# B&R Automation Studio project PLC code - cp (part 18)

#### MachineCtrl_Slow.st - Calling program actions
```iecst
PROGRAM _INIT

	versionPLC;

	IF gPLC.iVersion0<>gPermanentVersion.iVersion0 OR gPLC.iVersion1<>gPermanentVersion.iVersion1 OR gPLC.iVersion2<>gPermanentVersion.iVersion2 THEN
		gMachine.AutoCmd.xCleanModbus := TRUE;
	END_IF

	PLC_Init(ADR(gPLC));

END_PROGRAM

PROGRAM _CYCLIC

	// ACTIONS
	InternalPLC;

	VarsVersion;

	// Manage resetting PLC
	resetPLC;

	//Setting Serial Name of the PLC
	setSerialNumber;

	GeneralMachineData;

	//Devices parameters assignation not required to be executed in fast cycle
	OrdersPrinterSlow;

	// It allows CleanBelt action integrated on BeltManager
	IF gMachine.Pt.Clean.xCleanBeltWater THEN
		CleanBeltWater; //NOZOMITWO-1912
	ELSIF NOT gMachine.Pt.Clean.xCleanBeltForUv THEN
		CleanBelt;
	ELSE
		IF gMachine.Pt.MachineModel<>Type_CUBE AND gMachine.Pt.MachineModel<>Type_CUBE_GULLIVER AND gMachine.Pt.MachineModel<>Type_CUBE_INSPECTION AND gMachine.Pt.MachineModel<>Type_CUBE_GULLIVER_INSPECTION  THEN
			CleanBeltUv;
		END_IF
	END_IF

	//
	CleanBeltTop;

	// It allows to have consent line in belt orders
	//[RGP] Execute "ConsentsLine" always. It was previously called if "gBelt.parameters.xExistConsentLine" was active and always was
	ConsentsLine;

	// TOJMH: Review loop
	CleanSystem;

	BeltShot;

	PowerCtrl;
	SuctionBlower;
	ResetRouterAndCB;

	AirCleaner;

	AlarmsSlow;

	IF gMachine.Pt.MachineLights = MACHINE_LIGHTS_RGB THEN
		RgbLigths;
	ELSE
		LightBeacon;
	END_IF

	//[RGP] Execution of this action not conditioned to "xControlledByLine" so line has not to manage buzzer conditions defined inside printer as referencing block, starting belt...
	SoundBeacon;
	Air;
	JamSensors;

	ProgramsManager;

	Remote;

	// Check coherency of values and log possible mismatches
	CheckValues;

	//  Hw activation. Always sending the information from Sw
	// now added a parameter indicating if it is dynamically allowed to enable the system or not
	gDing.Parameters.xEnable := gMachine.parSw.Hw.xInstallThicknessSensor;
	gPhotoCells.parameters.xEnable := gMachine.parSw.Hw.xInstallnSensor;

	Startup;

	gMachine.St.xStarted := TRUE;
	gMachine.St.exec.slow := gMachine.St.exec.slow +1;

	//Powermeter assignation
	gPowermeters[1].Inputs.Comms.ReceivedDataModPowerMeter := gReceivedDataModPowerMeter1;
	gPowermeters[2].Inputs.Comms.ReceivedDataModPowerMeter := gReceivedDataModPowerMeter2;

END_PROGRAM
```

#### VersionPLC.st
```iecst
ACTION versionPLC:

    // PLC Version
	gPLC.iVersion0 := 23;    // Major version
	gPLC.iVersion1 := 68;    // Refactoring
	gPLC.iVersion2 := 394;   // Updated ExtPack
	gPLC.iVersion3 := 563;   // Version

END_ACTION
```

#### VarsVersion.st
```iecst
// THIS CODE IS AUTOGENERATED. DO NOT MODIFY IT WITH AUTOMATION STUDIO
// Generation: 10/07/2024 16:17:34
// Program version: 2.1.4.0

ACTION VarsVersion:

	gPLC.iVarsVersion0 := 9;
	gPLC.iVarsVersion1 := 42;
	gPLC.iVarsVersion2 := 1;
	gPLC.iVarsVersion3 := 2;

END_ACTION
```

- InternalPLC.st (reference to Logical/Printer/MachineCtrl/MachineCtrl_Slow/InternalPLC.st)

#### GeneralMachineData.st - Constant values according machine model
```iecst
ACTION GeneralMachineData:

	//////////////////////////////////////////////////////////////////////////////////////////////////////////////////////
	// BELT PARAMS      BELT PARAMS      BELT PARAMS      BELT PARAMS      BELT PARAMS      BELT PARAMS      BELT PARAMS
	// BELT PARAMS      BELT PARAMS      BELT PARAMS      BELT PARAMS      BELT PARAMS      BELT PARAMS      BELT PARAMS
	//////////////////////////////////////////////////////////////////////////////////////////////////////////////////////

	// Cleaning Belt limits cannot be lower than 1
	// Cleaning Belt parameters. Clean Belt disabled/enabled after delay
	iSPTilesToCleanBelt		:= MAX (gMachine.parSw.CleanBelt.iSPTilesToCleanBelt, MIN_TILES_FOR_CLEANING_BELT);
	iSPTilesToCleanBeltTop	:= MAX (gMachine.parSw.CleanBeltTop.iSPTilesToCleanBelt, MIN_TILES_FOR_CLEANING_BELT_TOP);

	////////// Belt Limits //////////////////////////////////
	//[RGP] Sending speed setpoint to gBelt. Not assigned directly from SW so maybe in the future SpeedSetpoint need to be used outside BeltPackage/BeltManager.
	//As done in previous lines by limiting maximum belt speed. //Not been able to have a Zero value in the SetPointSpeed
	gMachine.parSw.Safety.rMaxBeltSpeedSetPoint := MAX(gMachine.parSw.Safety.rMaxBeltSpeedSetPoint, 20); //At least a minimum value of 20.0m/min as max value

	//Belt speed definition
	IF gLine.StatusSummary.xEmptyingBelts THEN
		gBelt.parameters.rSetPointSpeed := MIN(gMachine.Pt.rBeltSpeedWhileEmptyBelt, gMachine.parSw.rBeltSpeedSetPoint);

	ELSIF gMachine.St.CleaningBelt.xCleaningProcessOnGoing THEN
		gBelt.parameters.rSetPointSpeed := INT_TO_REAL(gMachine.parSw.CleanBelt.iBeltSpeed);

	ELSIF (gLine.Status <> LINE_CONTROLLED_STOP AND gLine.Status <> LINE_CLEANINGPH AND gLine.Status <> LINE_STARTING_CLEANINGPH) OR NOT gMachine.Pt.xControlledByLine THEN
		gBelt.parameters.rSetPointSpeed := gMachine.parSw.rBeltSpeedSetPoint;
	END_IF

	// It gets belt direction following if machine configuration is left or right
	gBelt.parameters.Direction:= NOT gMachine.parSw.xMachineDirection;

	//Appling physical limitations
	IF NOT gMachine.Pt.xControlledByLine THEN
		gBelt.parameters.rMaxSpeed := gBelt.states.Hw.rMaxSpeed;
		gMachine.St.xDoubleLineAllowed := gMachine.Pt.Hw.xDoubleLineAllowed AND NOT gEdgeHoldDown.status.xEnabled;

	ELSE
		gBelt.parameters.rMaxSpeed := MIN(gBelt.states.Hw.rMaxSpeed, gLine.Parameters.Hw.rMaxSpeed);
		gMachine.St.xDoubleLineAllowed := gMachine.Pt.Hw.xDoubleLineAllowed AND gLine.Parameters.Hw.xDoubleLineAllowed AND NOT gEdgeHoldDown.status.xEnabled;
	END_IF

	////////////////////////////////////////////////////////////////////////////////////////////////////////////
	// BLOCK
	////////////////////////////////////////////////////////////////////////////////////////////////////////////

	xAnyBlockToPrint:=FALSE;
	FOR iIndexBlock:=1 TO gMachine.Pt.CT.iNumBlocks DO
		// It is used by ModeActive	implemented on printer
		IF gBlock[iIndexBlock].parSw.xEnableToPrint THEN
			xAnyBlockToPrint:=TRUE;
		END_IF
	END_FOR
	gMachine.St.Blocks.xAnyBlockToPrint:=xAnyBlockToPrint;

	///////////
	//White
	///////////
	IF gMachine.St.White.xInstalled THEN
		//Defining white bar index depending on machine direction. White is always first mechanically installed print bar
		IF gMachine.parSw.xMachineDirection THEN
			iWhiteBarMechanicalPosition := gBlock[1].parameters.Inks.iMaxMachinePrintBars;
		ELSE
			iWhiteBarMechanicalPosition := 1;
		END_IF

		IF NOT gMachine.St.White.xDebugMode THEN
			gMachine.St.White.xEnableToPrint := gInks[iWhiteBarMapping].status.xColorLoadedInJob;
		END_IF
	ELSE
		gMachine.St.White.xEnableToPrint := FALSE;
	END_IF

	///////////
	//Clear
	///////////
	IF gMachine.St.Clear.xInstalled THEN
		//Defining Primer bar index depending on machine direction. Primer is always first mechanically installed print bar
		IF gMachine.parSw.xMachineDirection THEN
			iPrimerBarMechanicalPosition := 3;
		ELSE
			iPrimerBarMechanicalPosition := 8;
		END_IF

		IF NOT gMachine.St.Clear.xDebugMode THEN
			gMachine.St.Clear.xEnableToPrint := gInks[iPrimerBarMapping].status.xColorLoadedInJob;
		END_IF

	ELSE
		gMachine.St.Clear.xEnableToPrint := FALSE;
	END_IF

	///////////
	//Color
	///////////
	IF NOT gMachine.St.Color.xDebugMode THEN
		//DELOREAN-3427: In case no color bar is loaded in job, curing led bar type CURING_APP_COLOR wont be activated
		xColorBarEnabledToPrint:=FALSE;
		FOR iIndexInks:=1 TO MAX_LAST_INK DO
			IF iIndexInks<>iWhiteBarMapping AND iIndexInks<>iPrimerBarMapping THEN
				IF gInks[iIndexInks].status.xColorLoadedInJob THEN
					xColorBarEnabledToPrint:=TRUE;
					EXIT;
				END_IF
			END_IF
		END_FOR
		gMachine.St.Color.xEnableToPrint := xColorBarEnabledToPrint;
	END_IF

	//CUBE-1197: due to this issue, protecting curing process by enabling curingled bar in case there is only one curing led bar.
	IF gMachine.Pt.Hw.iMaxCuringLedBars=1 THEN
		gMachine.St.Color.xEnableToPrint:=iIndexColorCuringLedBar=1;
		gMachine.St.Clear.xEnableToPrint :=iIndexPrimerCuringLedBar=1; //Pending to change the name of "iIndexPrimerCuringLedBar" by "iIndexClearCuringLedBar"
		xWhiteBarEnabledToPrint:=iIndexWhiteCuringLedBar=1;
	END_IF

	////////////////////////////////////////////////////////////////////////////////////////////////////////////
	// INKS >>>>> SLOW FOR		SLOW FOR		SLOW FOR		SLOW FOR		SLOW FOR
	////////////////////////////////////////////////////////////////////////////////////////////////////////////

	// Reset the index if the index is not valid. Just for protection. Never should enter here
	IF iIndexInksSlow = 0 OR iIndexInksSlow > MAX_LAST_INK THEN
		StartValuesForInksSlowFor;
		iIndexInksSlow := 1;
	END_IF

	IF gInks[iIndexInksSlow].status.xInksRunning THEN
		xAnyInkBarStarted := TRUE;
		IF rMaxStartedTempSetPoint < gInks[iIndexInksSlow].parSw.Temp.rSetPointTemp THEN
			rMaxStartedTempSetPoint := gInks[iIndexInksSlow].parSw.Temp.rSetPointTemp;
		END_IF
		IF rMaxStartedInkTemp < gInks[iIndexInksSlow].status.Temp.rTemp THEN
			rMaxStartedInkTemp:= gInks[iIndexInksSlow].status.Temp.rTemp;
		END_IF
		IF rMinStartedTempSetPoint > gInks[iIndexInksSlow].parSw.Temp.rSetPointTemp THEN
			rMinStartedTempSetPoint := gInks[iIndexInksSlow].parSw.Temp.rSetPointTemp;
		END_IF
		IF rMinStartedInkTemp > gInks[iIndexInksSlow].status.Temp.rTemp THEN
			rMinStartedInkTemp:= gInks[iIndexInksSlow].status.Temp.rTemp;
		END_IF

		//Any Tank Enabled
		IF gInks[iIndexInksSlow].status.xInkAndPreheatingRunning THEN
			xAnyTankHeaterEnabled:= TRUE;
		END_IF

		//Any bar printhead enabled
		IF gInks[iIndexInksSlow].signals.out.xOutPowPrintHead THEN
			xAnyPrintheadsPowered:= TRUE;
		END_IF

		//Depending on white bar mechanical position and if its enabled to print by electronics, status variable is set.
		//Cannot assume that gInks[1] will be the white bar so there is a case were white is physically installed but not defined in printer UI (disabled), gInks[1] then would be the following print bar assembled
		IF gInks[iIndexInksSlow].parSw.Config.iMappingBar = iWhiteBarMechanicalPosition THEN
			iWhiteBarMapping := iIndexInksSlow;
		ELSIF gInks[iIndexInksSlow].parSw.Config.iMappingBar = iPrimerBarMechanicalPosition THEN
			iPrimerBarMapping := iIndexInksSlow;
		END_IF

		IF gInks[iIndexInksSlow].parameters.InksChiller.iIndex > 0 AND gInks[iIndexInksSlow].parameters.InksChiller.iIndex < MAX_LAST_CHILLER THEN // Adding safety in the assignation
			gInks[iIndexInksSlow].parameters.InksChiller.Status := gChiller[gInks[iIndexInksSlow].parameters.InksChiller.iIndex].St.Status;
		END_IF

	END_IF

	IF gInks[iIndexInksSlow].parameters.PrintheadsChiller.iIndex > 0 AND gInks[iIndexInksSlow].parameters.PrintheadsChiller.iIndex < MAX_LAST_CHILLER THEN //Adding safety in the assignation
		gInks[iIndexInksSlow].parameters.PrintheadsChiller.Status := gChiller[gInks[iIndexInksSlow].parameters.PrintheadsChiller.iIndex].St.Status;
	END_IF

	iIndexInksSlow := iIndexInksSlow + 1;

	//If there is no logical bar with the mapping of the physical position, reset the outputs
	IF iIndexInksSlow > MAX_LAST_INK THEN

		//Assign data calculated to Machine Data
		gMachine.St.Inks.xAnyStarted := xAnyInkBarStarted;
		gMachine.St.Inks.rMaxTempSetPoint := rMaxStartedTempSetPoint;
		gMachine.St.Inks.rMinTempSetPoint := rMinStartedTempSetPoint;
		gMachine.St.Inks.rMaxTemp := rMaxStartedInkTemp;
		gMachine.St.Inks.rMinTemp := rMinStartedInkTemp;

		gMachine.St.Blocks.xAnyTankHeaterEnabled:= xAnyTankHeaterEnabled;
		gMachine.St.Blocks.xAnyPrintheadPowered:= xAnyPrintheadsPowered;

		StartValuesForInksSlowFor;
		iIndexInksSlow := 1;
	END_IF

	// Jetting Gap limits
	gMachine.parSw.rMarginPrint:= LIMIT(gMachine.Pt.CT.rMinMarginPrinting,gMachine.parSw.rMarginPrint,gMachine.Pt.CT.rMaxMarginPrinting);

	// Piece Tickness
	gMachine.parSw.Media.rThickness:= LIMIT(gMachine.Pt.CT.rMinTicknessMedia,gMachine.parSw.Media.rThickness,gMachine.Pt.CT.rMaxTicknessMedia);

	// Mounted Tile
	gMachine.parSw.Safety.rMountedPieceOverthickness:= LIMIT(gMachine.Pt.CT.rMinMountedPieceOverThick,gMachine.parSw.Safety.rMountedPieceOverthickness,gMachine.Pt.CT.rMaxMountedPieceOverThick);

	// Cleaning by pieces
	gMachine.parSw.Clean.iPiecesNumberToCleanL1:= MAX (gMachine.parSw.Clean.iPiecesNumberToCleanL1, GC_MIN_PIECES_TO_CLEAN);
	gMachine.parSw.Clean.iPiecesNumberToCleanL2:= MAX (gMachine.parSw.Clean.iPiecesNumberToCleanL2, GC_MIN_PIECES_TO_CLEAN);

	// Counters of shots printed by PD or by simulation
	//Counting out of any FOR. Makes no sense
	IF EDGEPOS (gMachine.St.ProductDetect.xProductDetectL1) THEN
		gMachine.Lg.udiPiecesCounterL1:= gMachine.Lg.udiPiecesCounterL1 + 1;
	END_IF

	IF EDGEPOS (gMachine.St.ProductDetect.xProductDetectL2) THEN
		gMachine.Lg.udiPiecesCounterL2:= gMachine.Lg.udiPiecesCounterL2 + 1;
	END_IF

	gMachine.St.xWorkingAsPBF := gMachine.parSw.Electronics.xIsPBF;

	//When entering in Working as PBF, modify diPiecesCounterStrobe to keep the same quantity of differences
	IF EDGEPOS(gMachine.St.xWorkingAsPBF) THEN
		gMachine.Lg.diPiecesCounterStrobe := gMachine.Lg.udiPiecesCounterL1 - gMachine.Lg.iDiffPiecesStrobeProductDetect;
	END_IF

	//Count strobes when Bit8 (strobe) is actived
	IF EDGEPOS(gMachine.In.iRelieve1>=256) AND gMachine.St.xWorkingAsPBF THEN
		gMachine.Lg.diPiecesCounterStrobe:= gMachine.Lg.diPiecesCounterStrobe + 1;
		gMachine.Out.iRelief1 := gMachine.In.iRelieve1;
	END_IF

	//Remove Relief output after time enough for the kernel to read it
	tofKeepReliefSignal.IN := EDGEPOS(gMachine.In.iRelieve1>=256) AND gMachine.St.xWorkingAsPBF;
	tofKeepReliefSignal.PT := t#900ms;
	tofKeepReliefSignal();
	IF NOT tofKeepReliefSignal.Q THEN
		gMachine.Out.iRelief1 := 0;
	END_IF

	//If Reset the counter, assign the value of Strobes to the value of PD
	IF gMachine.commands.xResetStrobePdDiff THEN
		gMachine.Lg.diPiecesCounterStrobe := gMachine.Lg.udiPiecesCounterL1;
		gMachine.Lg.iDiffPiecesStrobeProductDetect := 0;
		gMachine.commands.xResetStrobePdDiff := FALSE;
	END_IF
	IF EDGEPOS(gMachine.Lg.udiPiecesCounterL1 = 0) THEN
		gMachine.Lg.diPiecesCounterStrobe := - gMachine.Lg.iDiffPiecesStrobeProductDetect;
	END_IF

	//Define the diff counter. Updated just when receive a media in Product detect
	IF gMachine.St.xWorkingAsPBF AND EDGEPOS (gMachine.St.ProductDetect.xProductDetectL1) THEN
		gMachine.Lg.iDiffPiecesStrobeProductDetect := DINT_TO_INT(gMachine.Lg.udiPiecesCounterL1 - gMachine.Lg.diPiecesCounterStrobe);
	END_IF

	// Machine conversions
	gMachine.Lg.udiDifCounters:=ABS(UDINT_TO_INT(gMachine.Lg.udiPiecesCounterL1-gDing.State.diLgLowPieceCounter));

	//Enable degasser
	gMachine.Out.xDegasser:= gMachine.parSw.xDegasser AND NOT gMachine.Al.Warning.xAlrDegasserPressure;

	//Safety
	gSafetyController.Parameters.xSimulationMode := gMachine.Pt.ConfigNameID = GC_CONFIG_SIMTEST_ID;

	//Define a transmision data to do the first calculations and be receptive to next calculations
	DriveUnit.TransmissionData.TransmissionType := TRANS_LINEAL_PERIMETER;
	DriveUnit.TransmissionData.LinealPerimeter.PulsesPerTurn := GC_UNITS_BY_REV_DRIVE;
	DriveUnit.TransmissionData.LinealPerimeter.GearBox := 10.0;
	DriveUnit.TransmissionData.LinealPerimeter.Perimeter := 500.0;

	IF gThicknessCtrl.status.Belt.rBeltPositionMmInit<>rBeltPositionMmInitCopy THEN
		//Logger
		//Calculation of position when mounted media alarm is raised
		DriveUnit.pulsesDevice := gThicknessCtrl.status.Belt.rBeltPositionMmInit;
		DriveUnit.Calculation := CALC_POS_MM;
		DriveUnit();
		rBeltPositionMmInit := DriveUnit.PositionDevice;

		//Calculation of position when mounted media alarm is raised
		DriveUnit.PulsesSpeedDevice := gThicknessCtrl.status.Belt.rBeltSpeed;
		DriveUnit.Calculation := CALC_SPEED_MMIN;
		DriveUnit();
		rBeltSpeedInit := ABS(DriveUnit.SpeedMminDevice);

		rBeltPositionMmInitCopy := gThicknessCtrl.status.Belt.rBeltPositionMmInit;
	END_IF

	IF gThicknessCtrl.status.Belt.rBeltPositionMmFinal<>rBeltPositionMmFinalCopy THEN
		//Calculation of position when belt stops
		DriveUnit.pulsesDevice := gThicknessCtrl.status.Belt.rBeltPositionMmFinal;
		DriveUnit.Calculation := CALC_POS_MM;
		DriveUnit();
		rBeltPositionMmFinal := DriveUnit.PositionDevice;

		rBeltPositionMmFinalCopy := gThicknessCtrl.status.Belt.rBeltPositionMmFinal;
	END_IF

	rBeltDistanceTravelledMm := rBeltPositionMmFinal - rBeltPositionMmInit;
	IF rBeltDistanceTravelledMm<>rBeltDistanceTravelledMmCopy THEN
		//Logging distance run by belt from mounted media event to be stopped
		LogBeltDistanceTravelledWhenMountedMedia;

		rBeltDistanceTravelledMmCopy := rBeltDistanceTravelledMm;
	END_IF

END_ACTION

ACTION StartValuesForInksSlowFor:
	xAnyInkBarStarted := FALSE;
	rMaxStartedTempSetPoint := 0.0; //To be sure to be decreased
	rMaxStartedInkTemp := 0.0; //To be sure to be decreased
	rMinStartedTempSetPoint := 100.0; //To be sure to be decreased
	rMinStartedInkTemp := 100.0; //To be sure to be decreased
	xAnyTankHeaterEnabled := FALSE;
	xAnyPrintheadsPowered := FALSE;
END_ACTION
```

#### CleanBelt.st - Clean belt order
```iecst
ACTION CleanBelt:

	///////////////////////////////////////////////////////////////////////////////////////////////////////////////////
	// General conditions to clean belt	when machine is in AUTOMATIC OR MANUAL MODES
	///////////////////////////////////////////////////////////////////////////////////////////////////////////////////

	//Cleaning Belt by time. When cleaning, the time is reseted
	tonCleaningByTime.IN:= gBelt.states.xRuningBelt AND gMachine.parSw.CleanBelt.xCleanBeltByTime AND NOT tonCleaningByTime.Q AND NOT xCleanBeltOrder AND gMachine.St.Mode.xAuto;
	tonCleaningByTime.PT := MAX(gMachine.parSw.CleanBelt.tiCleaningBeltByTime, MIN_TIME_FOR_CLEANING_BELT); // Time converted from minutes to miliseconds
	tonCleaningByTime();

	//Delay falling the tray to be sure no water is poured inside the machine
	tofCleaningTrayBelt.IN:=xCleanBeltOrder;
	tofCleaningTrayBelt.PT:=T#200MS;
	tofCleaningTrayBelt();

	//Delay pneumatic pump to avoid pouring water inside the machine
	tonCleanBelt.IN:= xCleanBeltOrder;
	tonCleanBelt.PT:=T#900ms;
	tonCleanBelt();

	//If the belt is not running, it is not possible to clean it
	IF NOT gBelt.states.xRuningBelt THEN
		gMachine.commands.CleanBelt := ResetCleanBeltCommands;
		xCleanBeltOrder := FALSE;
		RETURN;
	END_IF

	// Tiles counter
	IF gMachine.parSw.CleanBelt.xCleanBeltByTiles AND (EDGEPOS (gMachine.St.ProductDetect.xProductDetectL1) OR EDGEPOS(gMachine.St.ProductDetect.xProductDetectL2)) THEN
		gMachine.Lg.iTilesCounterToClean:= gMachine.Lg.iTilesCounterToClean+1;
	END_IF

	//Cleaning by tiles. When cleaning, number of tiles is reseted
	IF (gMachine.parSw.CleanBelt.xCleanBeltByTiles AND (gMachine.Lg.iTilesCounterToClean >= INT_TO_UINT(iSPTilesToCleanBelt)) AND gMachine.St.Mode.xAuto) THEN
		xCleaningBeltByTiles:= TRUE;
	END_IF

	// Force cleaning applying delay. Why clean continuous is same that condition than force clean?
	IF gMachine.parSw.CleanBelt.xCleanBeltForced THEN
		xCleanBeltForced:= TRUE;
		gMachine.parSw.CleanBelt.xCleanBeltForced := FALSE;
	END_IF

	IF tonCleaningByTime.Q THEN
		xCleaningBeltByTime:=TRUE;
	END_IF

	IF (gMachine.parSw.CleanBelt.xCleanBeltContinue AND gMachine.St.Mode.xAuto) THEN
		xCleanBeltContinue := TRUE;
	ELSE
		xCleanBeltContinue := FALSE;
	END_IF

	IF xCleaningBeltByTiles OR xCleaningBeltByTime OR xCleanBeltForced OR xCleanBeltContinue THEN
		xCleanBeltOrder:=TRUE;

		//Removed orders when cleaning
		xCleaningBeltByTiles:=FALSE;
		gMachine.Lg.iTilesCounterToClean:=0;
		xCleaningBeltByTime:=FALSE;
		xCleanBeltForced := FALSE;
	END_IF

	// Managing the duration of the belt cleaning
	tonCleaningBelt.IN:= xCleanBeltOrder;
	tonCleaningBelt.PT := MAX(gMachine.parSw.CleanBelt.tiCleaningBeltDuration, MIN_DURATION_CLEANING_BELT);
	tonCleaningBelt();

	IF (tonCleaningBelt.Q AND NOT(xCleanBeltContinue)) OR EDGENEG(xCleanBeltContinue) THEN
		xCleanBeltOrder:=FALSE;
	END_IF

	//////////////////////
	// OUTPUT management
	//////////////////////
	//Clean belt

	//Pneumatic
	gMachine.commands.CleanBelt.xPistonFlojet := tofCleaningTrayBelt.Q;
	gMachine.commands.CleanBelt.xCleanBeltPump := tonCleanBelt.Q;

END_ACTION

ACTION CleanBeltTop:

	IF NOT gMachine.Pt.Clean.xCleanBeltTopInstall OR NOT gBelt.states.xRuningBelt THEN
		xCleanBeltTopOrder						:= FALSE;
		RETURN;
	END_IF

	///////////////////////////////////////////////////////////////////////////////////////////////////////////////////
	// General conditions to clean belt	when machine is in AUTOMATIC OR MANUAL MODES
	///////////////////////////////////////////////////////////////////////////////////////////////////////////////////

	//Cleaning Belt by time. When cleaning, the time is reseted
	tonCleanBeltTopByTime.IN := gMachine.parSw.CleanBeltTop.xCleanBeltByTime AND NOT tonCleanBeltTopByTime.Q AND NOT xCleanBeltTopOrder AND gMachine.St.Mode.xAuto;
	tonCleanBeltTopByTime.PT := MAX(gMachine.parSw.CleanBeltTop.tiCleaningBeltByTime, MIN_TIME_FOR_CLEANING_TOP_BELT);
	tonCleanBeltTopByTime();

	// Tiles counter
	IF gMachine.parSw.CleanBeltTop.xCleanBeltByTiles AND (EDGEPOS (gMachine.St.ProductDetect.xProductDetectL1) OR EDGEPOS(gMachine.St.ProductDetect.xProductDetectL2)) THEN
		gMachine.Lg.iTilesCounterToCleanBeltTop:= gMachine.Lg.iTilesCounterToCleanBeltTop + 1;
	END_IF

	//Cleaning by tiles. When cleaning, number of tiles is reseted
	IF (gMachine.parSw.CleanBeltTop.xCleanBeltByTiles AND (gMachine.Lg.iTilesCounterToCleanBeltTop >= INT_TO_UINT(iSPTilesToCleanBeltTop)) AND gMachine.St.Mode.xAuto) THEN
		xCleaningBeltTopByTiles:= TRUE;
	END_IF

	// Force cleaning applying delay. Why clean continuous is same that condition than force clean?
	IF gMachine.parSw.CleanBeltTop.xCleanBeltForced THEN
		xCleanBeltTopForced:= TRUE;
		gMachine.parSw.CleanBeltTop.xCleanBeltForced := FALSE;
	END_IF

	IF tonCleanBeltTopByTime.Q THEN
		xCleaningBeltTopByTime:=TRUE;
	END_IF

	IF (gMachine.parSw.CleanBeltTop.xCleanBeltContinue AND gMachine.St.Mode.xAuto) THEN
		xCleanBeltTopContinue := TRUE;
	ELSE
		xCleanBeltTopContinue := FALSE;
	END_IF

	IF xCleaningBeltTopByTiles OR xCleaningBeltTopByTime OR xCleanBeltTopForced OR xCleanBeltTopContinue THEN
		xCleanBeltTopOrder:=TRUE;

		//Removed orders when cleaning
		xCleaningBeltTopByTiles:=FALSE;
		gMachine.Lg.iTilesCounterToCleanBeltTop:=0;
		xCleaningBeltTopByTime:=FALSE;
		xCleanBeltTopForced := FALSE;
	END_IF

	// Managing the duration of the belt cleaning
	tonCleaningBeltTop.IN:= xCleanBeltTopOrder;
	tonCleaningBeltTop.PT := MAX(gMachine.parSw.CleanBeltTop.tiCleaningBeltDuration, MIN_DURATION_CLEANING_BELT_TOP);
	tonCleaningBeltTop();

	IF (tonCleaningBeltTop.Q AND NOT(gMachine.parSw.CleanBeltTop.xCleanBeltContinue)) OR EDGENEG(gMachine.parSw.CleanBeltTop.xCleanBeltContinue) THEN
		xCleanBeltTopOrder:=FALSE;
	END_IF

	//////////////////////
	// OUTPUT management
	//////////////////////

	gMachine.commands.CleanBelt.xCleanBeltTopScraper:=xCleanBeltTopOrder AND NOT gMachine.Pt.Clean.xCleanBeltForUv;

END_ACTION
```

#### ConsentLine.st - Consent Line
```iecst
ACTION ConsentsLine:
		(*
		View OF the machine from the Operator side

		>>>>>> LeftHandMachine 					RightHandMachine <<<<<<<<
		(BK_A #1 >> BK_B #2)		LOGICAL			(BK_A #2 << BK_B #1)

			          ################-################
		L2	          ################-################     L2
		------        ################-################   -------
		L1	          ################-################     L1
			##########################-###########################
			##########################-###########################
			    ######################-#######################
			    ######################-#######################
			    ######################-#######################
			    ######################-#######################

			BLOCK A [1-physical]				BLOCK B [2-physical]

		*)

	///////////////////////////////////////////////////
	// Consents depending if double or simple line
	//////////////////////////////////////////////////
	xDoubleLineConsent:= 	( gMachine.parSw.Dtp.iModeLine1=GC_DTP_STOP OR gMachine.In.xConsentL1Ok ) AND
							( gMachine.parSw.Dtp.iModeLine2=GC_DTP_STOP OR gMachine.In.xConsentL2Ok ) AND
							( gMachine.parSw.Dtp.iModeLine1<>GC_DTP_STOP OR gMachine.parSw.Dtp.iModeLine2<>GC_DTP_STOP);

	tonDelayConsentInput.IN:= 	(NOT gMachine.parSw.Dtp.xDoubleLine AND gMachine.In.xConsentL1Ok ) OR
								(gMachine.parSw.Dtp.xDoubleLine AND xDoubleLineConsent );
	tonDelayConsentInput.PT:= T#500ms;
	tonDelayConsentInput();

	gMachine.St.Consent.xConsent:= tonDelayConsentInput.Q;

	//Raise Bars without consent
	xAvoidRaiseBarsNotConsent := gMachine.Al.Alarm.xAlarmNotInPrintPosition OR gMachine.Al.Warning.xNotLoadedImage;
	tonUpBarsNoConsent.IN :=	gMachine.St.AutoMode.xProduction AND NOT xAvoidRaiseBarsNotConsent AND NOT gMachine.St.Consent.xConsent;
	tonUpBarsNoConsent.PT:= T#5m;
	tonUpBarsNoConsent();
	gMachine.St.Consent.xUpWithNoConsentCountingTime := tonUpBarsNoConsent.IN;

	//Split the assignation to allow an external assignation from simulation to avoid waiting 5min
	IF EDGEPOS(tonUpBarsNoConsent.Q) THEN
		gMachine.St.Consent.xUpWithNoConsent := TRUE;
	END_IF
	IF NOT gMachine.St.AutoMode.xProduction OR EDGEPOS(gMachine.St.Position.xInPrint) THEN
		gMachine.St.Consent.xUpWithNoConsent := FALSE;
	END_IF

	IF gMachine.St.Consent.xUpWithNoConsent OR gMachine.St.xProtectBendedWithPause THEN
		gMachine.St.Consent.xOrderToEmpyBelt := TRUE;
	ELSIF NOT gThicknessCtrl.status.MediaPosition.xMediaInside THEN
		gMachine.St.Consent.xOrderToEmpyBelt := FALSE;
	END_IF

	///////////////////////////////////////////////////////////////////////////////////////
	///////////////////////////////////////////////////////////////////////////////////////
	///////////////////////////////////////////////////////////////////////////////////////

	// Pending to test
	//Consent Outputs for L1
	//Single line L1, When belt is runing is because we had consent
	xOutputConsentInSingleLineL1:=	NOT gMachine.parSw.Dtp.xDoubleLine AND
									gMachine.In.xConsentL1Ok AND
									gMachine.St.AutoMode.xProdORByPass AND
									NOT gThicknessCtrl.status.MediaPosition.xMountedMediaInside AND
									NOT gMachine.St.Blocks.xBlockAlarmToEmpyBelt AND
									NOT gMachine.St.Consent.xOrderToEmpyBelt;

	xOutputConsentInByPassL1 := gMachine.St.AutoMode.xBypass AND
								gMachine.In.xConsentL1Ok AND
								(NOT gMachine.parSw.Dtp.xDoubleLine OR (gMachine.parSw.Dtp.xDoubleLine AND gMachine.parSw.Dtp.iModeLine1<>GC_DTP_STOP)) ;
	xOutputConsentInByPassL2 := gMachine.St.AutoMode.xBypass AND
								gMachine.In.xConsentL2Ok AND
								gMachine.parSw.Dtp.xDoubleLine AND gMachine.parSw.Dtp.iModeLine2<>GC_DTP_STOP ;

	xOutputConsentInDTPL1:=	gMachine.St.AutoMode.xProdORByPass AND
							NOT gMachine.St.Blocks.xBlockAlarmToEmpyBelt AND
							(gMachine.parSw.Dtp.xDoubleLine AND gMachine.parSw.Dtp.iModeLine1<>GC_DTP_STOP);
	xOutputConsentInDTPL2:=	gMachine.St.AutoMode.xProdORByPass AND
							NOT gMachine.St.Blocks.xBlockAlarmToEmpyBelt AND
							(gMachine.parSw.Dtp.xDoubleLine AND gMachine.parSw.Dtp.iModeLine2<>GC_DTP_STOP);

	//Consider the delay of the output signal configured in SW
	tonDelayConsentOutL1.IN:= gBelt.states.xRuningBelt AND (xOutputConsentInSingleLineL1 OR xOutputConsentInDTPL1 OR xOutputConsentInByPassL1);// It checked in both single or dtpL1
	tonDelayConsentOutL1.PT:= gMachine.parSw.tiDelayConsent;
	tonDelayConsentOutL1();
	tonDelayConsentOutL2.IN:= gBelt.states.xRuningBelt AND (xOutputConsentInDTPL2 OR xOutputConsentInByPassL2);
	tonDelayConsentOutL2.PT:= gMachine.parSw.tiDelayConsent;
	tonDelayConsentOutL2();

	gMachine.Out.xConsentL1:= tonDelayConsentOutL1.Q;
	gMachine.Out.xConsentL2:= tonDelayConsentOutL2.Q;

	////////////////////////////
	// COMPENSERS
	////////////////////////////
	gMachine.Out.xCompenserLine1:= gMachine.commands.xCompenserLine1;
	gMachine.Out.xCompenserLine2:= gMachine.commands.xCompenserLine2;

END_ACTION
```

#### OrdersPrinterSlow.st
```iecst
ACTION OrdersPrinterSlow:

	// GENERAL MACHINE
	gMachine.St.Consent.xLackOfConsent := gBelt.states.State = BELT_NOT_CONSENT; //With run order but without consent

	///////////////////////////////////////////////////////////////////////////////////
	///////////////////////////////////////////////////////////////////////////////////
	/////////////   BLOCK BLOCK BLOCK BLOCK BLOCK BLOCK BLOCK      ////////////////////
	/////////////   BLOCK BLOCK BLOCK BLOCK BLOCK BLOCK BLOCK      ////////////////////
	///////////////////////////////////////////////////////////////////////////////////
	///////////////////////////////////////////////////////////////////////////////////

	FOR iIndexBlock:=GC_FIRST_BLOCK TO gMachine.Pt.CT.iNumBlocks DO
		// Double Line
		gBlock[iIndexBlock].Out.xEnableDobleShot:= gMachine.parSw.Dtp.xDoubleLine;

		// Vertical motor
		IF gMachine.Pt.xDynamicPrePrintingPos THEN
			IF NOT gEdgeHoldDown.status.xEnabled THEN
				IF gPhotoCells.status.xInstalled THEN
					gBlock[iIndexBlock].parameters.rPrePrintingPos := gThicknessCtrl.status.Heigh.rMediaThickness + gPhotoCells.status.rOffsetToMounted;
				ELSIF gDing.State.xDingInstalled THEN
					gBlock[iIndexBlock].parameters.rPrePrintingPos := gThicknessCtrl.status.Heigh.rMediaThickness  + gDing.Parameters.rOverThicknessToMounted;
				END_IF
			ELSE
				gBlock[iIndexBlock].parameters.rPrePrintingPos := gEdgeHoldDown.status.rBlockPrePrintingPosition;
			END_IF
		END_IF

		// Clean Motor
		gBlock[iIndexBlock].parameters.Icla.iCleanMotorSpeedBwd:=gMachine.parSw.Clean.iCleanMotorSpeedBwd;
		gBlock[iIndexBlock].parameters.Icla.iCleanMotorSpeedFwd:=gMachine.parSw.Clean.iCleanMotorSpeedFwd;

		//Icla action
		gBlock[iIndexBlock].parameters.Icla.rMinPrintHeadPos	:= gMachine.Pt.rMinPrintHeadPos;
		gBlock[iIndexBlock].parameters.Icla.rLastHeadPosition	:= LIMIT(gMachine.Pt.rMinPrintHeadPos, gMachine.parSw.rLastHeadPosition, gMachine.Pt.rMaxPrintHeadPos);
		gBlock[iIndexBlock].parameters.Icla.rFirstHeadPosition	:= LIMIT(gMachine.Pt.rMinPrintHeadPos, gMachine.parSw.rFirstHeadPosition, gBlock[iIndexBlock].parameters.Icla.rLastHeadPosition);

		//Icla movement
		gBlock[iIndexBlock].parameters.Icla.rPositionCleanMotorFwd	:= gBlock[iIndexBlock].parameters.Icla.rLastHeadPosition;

		gBlock[iIndexBlock].parameters.uiCleaningType 			:= INT_TO_USINT(gMachine.parSw.Clean.iCleaningType);

	END_FOR

	//ANALOG THICKNESS CONTROL
	gDing.Parameters.rMachineMinTicknessMedia := gMachine.Pt.CT.rMinTicknessMedia;
	gDing.Parameters.rMountedMediaLevelInBypassMode := gMachine.Pt.CT.rMountedMediaLevelInBypassMode;
	gDing.Parameters.xSimulationMode := gMachine.Pt.ConfigNameID = GC_CONFIG_SIMTEST_ID;

	//THICKNESS DETECTION
	gThicknessCtrl.parameters.Belt.rMinBeltSpeedToStart 	:= gc_rMinSpeedToStart;
	gThicknessCtrl.parameters.Cure.White.xEnabled			:= gCuringLed[iIndexWhiteCuringLedBar].Parameters.xInstalled; // Enable can be changed dynamically and tracking is needed always is installed
	gThicknessCtrl.parameters.Cure.White.iStartWindow		:= MAX(gCuringLed[iIndexWhiteCuringLedBar].Parameters.iCuringPosition - gCuringLed[iIndexWhiteCuringLedBar].parSw.iPreCuringOffset, 0); //If not limited, considered the negative as maximum and do not cure
	gThicknessCtrl.parameters.Cure.White.iEndWindow			:= gCuringLed[iIndexWhiteCuringLedBar].Parameters.iCuringPosition + (gCuringLed[iIndexWhiteCuringLedBar].Parameters.iCuringWindow/10) + gCuringLed[1].parSw.iPostCuringOffset;
	gThicknessCtrl.parameters.Cure.Color.xEnabled			:= gCuringLed[iIndexColorCuringLedBar].Parameters.xInstalled; // Enable can be changed dynamically and tracking is needed always is installed
	gThicknessCtrl.parameters.Cure.Color.iStartWindow		:= MAX(gCuringLed[iIndexColorCuringLedBar].Parameters.iCuringPosition - gCuringLed[iIndexColorCuringLedBar].parSw.iPreCuringOffset, 0); //If not limited, considered the negative as maximum and do not cure
	gThicknessCtrl.parameters.Cure.Color.iEndWindow			:= gCuringLed[iIndexColorCuringLedBar].Parameters.iCuringPosition + (gCuringLed[iIndexColorCuringLedBar].Parameters.iCuringWindow/10) + gCuringLed[iIndexColorCuringLedBar].parSw.iPostCuringOffset;
	gThicknessCtrl.parameters.Cure.Primer.xEnabled			:= gCuringLed[iIndexPrimerCuringLedBar].Parameters.xInstalled; // Enable can be changed dynamically and tracking is needed always is installed
	gThicknessCtrl.parameters.Cure.Primer.iStartWindow		:= MAX(gCuringLed[iIndexPrimerCuringLedBar].Parameters.iCuringPosition - gCuringLed[iIndexPrimerCuringLedBar].parSw.iPreCuringOffset, 0); //If not limited, considered the negative as maximum and do not cure
	gThicknessCtrl.parameters.Cure.Primer.iEndWindow		:= gCuringLed[iIndexPrimerCuringLedBar].Parameters.iCuringPosition + (gCuringLed[iIndexPrimerCuringLedBar].Parameters.iCuringWindow/10) + gCuringLed[iIndexColorCuringLedBar].parSw.iPostCuringOffset;

	gThicknessCtrl.parameters.Cure.xEnableTracking			:= gMachine.Pt.Hw.iMaxCuringLedBars>0;

	// Till now just considering Line 1
	gThicknessCtrl.parameters.ContinuousMedia.MediaData.iLine := 1;
	gThicknessCtrl.parameters.ContinuousMedia.MediaData.rThickness := gMachine.parSw.Media.rThickness;
	gThicknessCtrl.parameters.ContinuousMedia.MediaData.rWidth := gMachine.parSw.Media.rWidth;
	gThicknessCtrl.parameters.ContinuousMedia.MediaData.rLength := gMachine.parSw.Media.rLength;
	gThicknessCtrl.parameters.ContinuousMedia.MediaData.rCrossOffset := gMachine.parSw.Media.rOffsetRegisterL1;
	IF gMachine.Pt.ConfigNameID<> GC_CONFIG_SIMTEST_ID THEN
		gThicknessCtrl.parameters.ContinuousMedia.MediaData.xHasWhite := gMachine.St.White.xEnableToPrint;
		gThicknessCtrl.parameters.ContinuousMedia.MediaData.xHasClear := gMachine.St.Clear.xEnableToPrint;
	ELSE
		gThicknessCtrl.parameters.ContinuousMedia.MediaData.xHasWhite := gCuringLed[iIndexWhiteCuringLedBar].Parameters.xInstalled;
		gThicknessCtrl.parameters.ContinuousMedia.MediaData.xHasClear := gCuringLed[iIndexPrimerCuringLedBar].Parameters.xInstalled;
	END_IF
	gThicknessCtrl.parameters.ContinuousMedia.MediaData.rDocWidth := gMachine.parSw.Document.rWidth;
	gThicknessCtrl.parameters.ContinuousMedia.MediaData.rDocLength := gMachine.parSw.Document.rLength;
	gThicknessCtrl.parameters.ContinuousMedia.MediaData.rDocCrossOffset := gMachine.parSw.Document.rOffsetL1;

	gThicknessCtrl.parameters.xDoubleLine := gMachine.parSw.Dtp.xDoubleLine;
	gThicknessCtrl.parameters.Detection.Array.xEnableSensorIncoherAlarm := gPhotoCells.status.xTrustPhotocellASignal;

	CASE gStacker.Status.StackerType OF
		//Full stacker requires to set reject order (digital output) when boards "tail" is just about to exit printer's belt
		STACKERTY_FULL_S,
		STACKERTY_UNDEFINED:
			gThicknessCtrl.parameters.Reject.RejectBoardEdge := REJECT_REAR;

		//Bundle stacker requires to set reject order (digital output) when boards "head" is just about to exit printer's belt
		STACKERTY_BUNDLE_S:
			gThicknessCtrl.parameters.Reject.RejectBoardEdge := REJECT_FRONT;
	END_CASE

	//CURING LAMPS
	FOR iIndexCuringLed:=1 TO MAX_LAST_CURING_LED DO

		IF gMachine.Pt.Cure.xForceMaxWidth THEN
			gCuringLed[iIndexCuringLed].Parameters.iMediaWidth 		:= gMachine.Pt.Hw.iWidth;
			gCuringLed[iIndexCuringLed].Parameters.iDocumentWidth 	:= gMachine.Pt.Hw.iWidth;
			gCuringLed[iIndexCuringLed].Parameters.iMediaOffsetL1 	:= (-1) * gMachine.Pt.Hw.iWidth / 2;
			gCuringLed[iIndexCuringLed].Parameters.iDocumentOffsetL1:= gCuringLed[iIndexCuringLed].Parameters.iMediaOffsetL1;
			gCuringLed[iIndexCuringLed].Parameters.iMediaOffsetL2 	:= gCuringLed[iIndexCuringLed].Parameters.iMediaOffsetL1;
			gCuringLed[iIndexCuringLed].Parameters.iDocumentOffsetL2:= gCuringLed[iIndexCuringLed].Parameters.iMediaOffsetL1;
		ELSE
			gCuringLed[iIndexCuringLed].Parameters.iMediaWidth 		:= REAL_TO_UINT(gMachine.parSw.Media.rWidth);
			gCuringLed[iIndexCuringLed].Parameters.iDocumentWidth 	:= REAL_TO_UINT(gMachine.parSw.Document.rWidth);
			gCuringLed[iIndexCuringLed].Parameters.iMediaOffsetL1 	:= REAL_TO_INT(gMachine.parSw.Media.rOffsetRegisterL1);
			gCuringLed[iIndexCuringLed].Parameters.iDocumentOffsetL1:= REAL_TO_INT(gMachine.parSw.Document.rOffsetL1);
			gCuringLed[iIndexCuringLed].Parameters.iMediaOffsetL2 	:= REAL_TO_INT(gMachine.parSw.Media.rOffsetRegisterL2);
			gCuringLed[iIndexCuringLed].Parameters.iDocumentOffsetL2:= REAL_TO_INT(gMachine.parSw.Document.rOffsetL2);
		END_IF

		gCuringLed[iIndexCuringLed].Parameters.xDoubleLine 		:= gMachine.parSw.Dtp.xDoubleLine AND gMachine.Pt.Hw.xDoubleLineAllowed;

		gCuringLed[iIndexCuringLed].Parameters.rBeltCurrentSpeed:= gBelt.states.rCurrentSpeed;
		gCuringLed[iIndexCuringLed].Parameters.Mode 			:= gMachine.St.Mode;
		gCuringLed[iIndexCuringLed].Parameters.xCureBySpeed		:= gMachine.parSw.Curing.xCureBySpeed;
		gCuringLed[iIndexCuringLed].Parameters.xCureByStretch	:= gMachine.parSw.Curing.xCureByStretch AND gMachine.Pt.Cure.xCuringByStretchAllowed;
		gCuringLed[iIndexCuringLed].Parameters.xOptimizeCuring	:= gMachine.parSw.Curing.xOptimizeCuring OR gEdgeHoldDown.status.xEnabled;;
		gCuringLed[iIndexCuringLed].Parameters.xSimulationMode	:=  gMachine.Pt.ConfigNameID = GC_CONFIG_SIMTEST_ID;

		//Setting max curing variables depending on EdgeHoldDown
		IF  gEdgeHoldDown.status.xEnabled THEN
			gCuringLed[iIndexCuringLed].Parameters.iMaxCuringAreaWidth := REAL_TO_UINT(gMachine.parSw.Media.rWidth-2*gEdgeHoldDown.parSw.iOverlap-2*gCuringLed[iIndexCuringLed].Parameters.iSlmWidth);
			gCuringLed[iIndexCuringLed].Parameters.iMaxCuringAreaOffsetL1 := REAL_TO_INT(gCuringLed[iIndexCuringLed].Parameters.iMaxCuringAreaWidth/2)*(-1);
			gCuringLed[iIndexCuringLed].Parameters.iMaxCuringAreaOffsetL2 := REAL_TO_INT(gCuringLed[iIndexCuringLed].Parameters.iMaxCuringAreaWidth/2);
		ELSE
			gCuringLed[iIndexCuringLed].Parameters.iMaxCuringAreaWidth := gMachine.Pt.Hw.iWidth;
			gCuringLed[iIndexCuringLed].Parameters.iMaxCuringAreaOffsetL1 := REAL_TO_INT(gMachine.Pt.Hw.iWidth/2)*(-1);
			gCuringLed[iIndexCuringLed].Parameters.iMaxCuringAreaOffsetL2 := REAL_TO_INT(gMachine.Pt.Hw.iWidth/2);
		END_IF

	END_FOR

	IF gMachine.St.White.xEnableToPrint THEN
		gCuringLed[iIndexWhiteCuringLedBar].Parameters.xEnabled := TRUE;
	ELSIF gThicknessCtrl.status.Belt.xBeltEmpty THEN
		gCuringLed[iIndexWhiteCuringLedBar].Parameters.xEnabled := FALSE;
	END_IF

	IF gMachine.Pt.CT.iNumCuringLeds = 1 OR gMachine.St.Color.xEnableToPrint THEN
		gCuringLed[iIndexColorCuringLedBar].Parameters.xEnabled := TRUE;
	ELSIF gThicknessCtrl.status.Belt.xBeltEmpty THEN
		gCuringLed[iIndexColorCuringLedBar].Parameters.xEnabled := FALSE;
	END_IF

	IF gMachine.St.Clear.xEnableToPrint THEN
		gCuringLed[iIndexPrimerCuringLedBar].Parameters.xEnabled := TRUE;
	ELSIF gThicknessCtrl.status.Belt.xBeltEmpty THEN
		gCuringLed[iIndexPrimerCuringLedBar].Parameters.xEnabled := FALSE;
	END_IF

	IF NOT gMachine.Pt.xControlledByLine THEN
		gMachine.Pt.Media.iMaxMediaWidth := gMachine.Pt.Hw.iWidth;
		gMachine.Pt.Media.iMaxMediaLength := gMachine.parSw.Hw.iMaxMediaLength;
		gMachine.Pt.Media.iMinMediaWidth := 300;
		gMachine.Pt.Media.iMinMediaLength := 300;
		gMachine.Pt.Media.rMaxMediaThickness := gMachine.Pt.CT.rMaxTicknessMedia;
		gMachine.Pt.Media.rMinMediaThickness := gMachine.Pt.CT.rMinTicknessMedia;
	END_IF

	// Printer remotelly controlled
	IF EDGENEG(gMachine.St.AutoMode.xStop) OR EDGENEG(gMachine.St.Mode.xAuto) OR gMachine.St.Mode.xZero THEN
		//To avoid start blowers when returning to Auto.Stop
		gMachine.commands.Remote.xStartBlowers := FALSE;
	END_IF

	//CHILLER
	IF iIndexChillersSlow=0 OR iIndexChillersSlow> gMachine.Pt.Hw.iMaxNumChillers THEN
		iIndexChillersSlow:=1;
	END_IF

	IF gChiller[iIndexChillersSlow].Parameters.xInstalled THEN
		xRunChiller := FALSE;
		//Review printheads conditions to run its chiller
		FOR iIndexInks:=1 TO MAX_LAST_INK DO
			IF gInks[iIndexInks].parameters.PrintheadsChiller.iIndex = iIndexChillersSlow THEN
				IF gInks[iIndexInks].signals.out.xOutPowPrintHead THEN
					xRunChiller := TRUE;
				END_IF
			END_IF
		END_FOR

		//Review inks conditions to run its chiller
		FOR iIndexInks:=1 TO MAX_LAST_INK DO
			IF gInks[iIndexInks].parameters.InksChiller.iIndex = iIndexChillersSlow THEN
				IF gInks[iIndexInks].status.xInksRunning THEN
					xRunChiller := TRUE;
				END_IF
			END_IF
		END_FOR

		//Review curing led bars conditions to run its chiller
		FOR iIndexCuringLed:=1 TO MAX_LAST_CURING_LED DO
			IF gCuringLed[iIndexCuringLed].Parameters.iChillerIndex = iIndexChillersSlow THEN
				IF gCuringLed[iIndexCuringLed].Signals.Outputs.xRunChiller THEN
					xRunChiller := TRUE;
				END_IF
			END_IF
		END_FOR

		gChiller[iIndexChillersSlow].Orders.xRun := xRunChiller;

	END_IF

	iIndexChillersSlow:=iIndexChillersSlow+1;

	//Antistatic device
	gMachine.Out.xAntiStaticPOn := gMachine.St.Position.xInPrint;

	//Commands
	FOR iIndex:=1 TO gMachine.Pt.Hw.iMaxNumChillers DO
		gChiller[iIndex].commands.xMute	:= gMachine.AutoCmd.xMuteAlarms;
		gChiller[iIndex].commands.xReset		:= gMachine.AutoCmd.xReset;
	END_FOR

	//Powermeters
	FOR iIndex:=1 TO gMachine.Pt.Hw.iMaxNumPowerMeters DO
		IF gPowermeters[iIndex].Parameters.xInstalled THEN
			gPowermeters[iIndex].Commands.xMute	:= gMachine.AutoCmd.xMuteAlarms;
			gPowermeters[iIndex].Commands.xReset:= gMachine.AutoCmd.xReset;
		END_IF
	END_FOR

END_ACTION
```

#### Remote.st
```iecst
ACTION Remote:

	gMachine.St.Remote.xMachineReady := gBelt.states.xRuningBelt AND gTransVacuum[1].Status.Blower.xMoving AND NOT gMachine.In.xRemoteJog;
	gMachine.St.Remote.xReadyToJogInJamRecovery := gMachine.St.AutoMode.xJamRecovery AND gBlock[1].Status.Position.xInPrint AND gTransVacuum[1].Status.Blower.xMoving;

	iReasonReadyToReset := 16#FFFF;
	iReasonReadyToReset.0 := gSafetyController.Inputs.xPrinterBacksideEstop;
	iReasonReadyToReset.1 := gSafetyController.Inputs.xPrinterFrontsideEstop;
	iReasonReadyToReset.2 := gSafetyController.Inputs.xFeederEstop;
	iReasonReadyToReset.3 := gSafetyController.Inputs.xPrimerEstop;
	iReasonReadyToReset.4 := gSafetyController.Inputs.xOvervarnishEstop;
	iReasonReadyToReset.5 := gSafetyController.Inputs.xStackerEstop;
	iReasonReadyToReset.6 := gSafetyController.Inputs.xPrinterLightCurtain;
	iReasonReadyToReset.7 := gSafetyController.Inputs.xPrinterDoorLock;

	gMachine.St.Remote.xSafetyReadyToReset := iReasonReadyToReset = 16#FFFF;

END_ACTION
```

#### EventLog.st
```iecst
ACTION LogWarningSize:

	stEventLogWarningSize.Source := ELOG_TYPE_GENERAL;
	stEventLogWarningSize.Severity:= ELOG_SEVERITY_WARNING;
	stEventLogWarningSize.Facility:= 0;
	stEventLogWarningSize.ErrorCode:=0;

	stEventLogWarningSize.Text := 'Mismatch in Media values. ';

	//Adding nState data to log
	strAuxEventDesc := '. Width= ';
	brsstrcat(ADR(stEventLogWarningSize.Text), ADR(strAuxEventDesc));
	brsitoa(REAL_TO_INT(gMachine.parSw.Media.rWidth), ADR(strAuxEventDesc));
	brsstrcat(ADR(stEventLogWarningSize.Text), ADR(strAuxEventDesc));
	strAuxEventDesc := '. OffsetL1= ';
	brsstrcat(ADR(stEventLogWarningSize.Text), ADR(strAuxEventDesc));
	brsitoa(REAL_TO_INT(gMachine.parSw.Media.rOffsetRegisterL1), ADR(strAuxEventDesc));
	brsstrcat(ADR(stEventLogWarningSize.Text), ADR(strAuxEventDesc));

	gEventLogLoader(EventData := ADR(stEventLogWarningSize));

END_ACTION

ACTION LogImageLoadedL1:

	stEventLogImgLoadedL1.Source := ELOG_TYPE_GENERAL;
	stEventLogImgLoadedL1.Severity:= ELOG_SEVERITY_INFO;
	stEventLogImgLoadedL1.Facility:= 0;
	stEventLogImgLoadedL1.ErrorCode:=0;

	stEventLogImgLoadedL1.Text := 'Image loaded L1';

	gEventLogLoader(EventData := ADR(stEventLogImgLoadedL1));

END_ACTION

ACTION LogImageUnLoadedL1:

	stEventLogImgUnLoadedL1.Source := ELOG_TYPE_GENERAL;
	stEventLogImgUnLoadedL1.Severity:= ELOG_SEVERITY_INFO;
	stEventLogImgUnLoadedL1.Facility:= 0;
	stEventLogImgUnLoadedL1.ErrorCode:=0;

	stEventLogImgUnLoadedL1.Text := 'Image Unloaded L1';

	gEventLogLoader(EventData := ADR(stEventLogImgUnLoadedL1));

END_ACTION

ACTION LogAlarmImageNotLoaded:

	stEventLogAlrNotLoadedImage.Source := ELOG_TYPE_GENERAL;
	stEventLogAlrNotLoadedImage.Severity:= ELOG_SEVERITY_INFO;
	stEventLogAlrNotLoadedImage.Facility:= 0;
	stEventLogAlrNotLoadedImage.ErrorCode:=0;

	stEventLogAlrNotLoadedImage.Text := 'Alarm Image NOT loaded';

	gEventLogLoader(EventData := ADR(stEventLogAlrNotLoadedImage));

END_ACTION

ACTION LogAlarmImageLoadedButNoInkBarRelated:

	stLogAlrImageLoadButNoBarRelated.Source := ELOG_TYPE_GENERAL;
	stLogAlrImageLoadButNoBarRelated.Severity:= ELOG_SEVERITY_INFO;
	stLogAlrImageLoadButNoBarRelated.Facility:= 0;
	stLogAlrImageLoadButNoBarRelated.ErrorCode:=0;

	stLogAlrImageLoadButNoBarRelated.Text := 'Alarm Image loaded but no ink bar status has color loaded';

	gEventLogLoader(EventData := ADR(stLogAlrImageLoadButNoBarRelated));

END_ACTION

ACTION LogBeltDistanceTravelledWhenMountedMedia:
	stEventLogBeltDistanceTravelled.Source := ELOG_TYPE_DETECTION;
	stEventLogBeltDistanceTravelled.Severity:= ELOG_SEVERITY_INFO;
	stEventLogBeltDistanceTravelled.Facility:= 0;
	stEventLogBeltDistanceTravelled.ErrorCode:=0;
	stEventLogBeltDistanceTravelled.Text := 'Belt distance travelled: ';

	brsftoa(rBeltDistanceTravelledMm, ADR(strAuxEventDesc));
	brsstrcat(ADR(stEventLogBeltDistanceTravelled.Text), ADR(strAuxEventDesc));

	brsstrcat(ADR(stEventLogBeltDistanceTravelled.Text), ADR('mm at '));
	brsftoa(rBeltSpeedInit, ADR(strAuxEventDesc));
	brsstrcat(ADR(stEventLogBeltDistanceTravelled.Text), ADR(strAuxEventDesc));

	brsstrcat(ADR(stEventLogBeltDistanceTravelled.Text), ADR('mm/min. Decel at  '));
	brsftoa(gBelt.states.rDeceleration, ADR(strAuxEventDesc));
	brsstrcat(ADR(stEventLogBeltDistanceTravelled.Text), ADR(strAuxEventDesc));

	brsstrcat(ADR(stEventLogBeltDistanceTravelled.Text), ADR('mm/s2. Vacuum pressure:'));
	brsftoa(gTransVacuum[1].Status.rPressurePerc, ADR(strAuxEventDesc));
	brsstrcat(ADR(stEventLogBeltDistanceTravelled.Text), ADR(strAuxEventDesc));

	brsstrcat(ADR(stEventLogBeltDistanceTravelled.Text), ADR('%. Blowers DC:'));
	brsftoa(gTransVacuum[1].Status.Blower.rDutyCycle, ADR(strAuxEventDesc));
	brsstrcat(ADR(stEventLogBeltDistanceTravelled.Text), ADR(strAuxEventDesc));
	brsstrcat(ADR(stEventLogBeltDistanceTravelled.Text), ADR('%'));

	gEventLogLoader(EventData := ADR(stEventLogBeltDistanceTravelled));

END_ACTION
```

- MachineCtrlConsentStates.graphml - Machine states ctrl (not shown)

### Package Logical/Printer/PhysicalMapping - Physical inputs assignation

### Program Logical/Printer/PhysicalMapping/PhysicalMapInputs (IEC)

#### InputsS1400.st - PhysicalInputs
```iecst
ACTION InputsS1400:

	(* CABINET 01 *)

	// X20DIF371_001

	// gMachine.In.iMachineModelCode assigned in an specific Action

	gMachine.In.Buttons.xStart					:= X20DIF371_001.DInput[7];
	gMachine.In.Buttons.xStop					:= NOT X20DIF371_001.DInput[8];
	gMachine.In.Buttons.xAuto					:= X20DIF371_001.DInput[9];
	gMachine.In.Buttons.xZero					:= NOT X20DIF371_001.DInput[10];
	gMachine.In.Buttons.xManual					:= X20DIF371_001.DInput[11];
	//gMachine.In.Buttons.xReset					:= X20DIF371_001.DInput[12];
	gMachine.In.ProductDetect.pPDCarriageSignalL1 := ADR(X20DIF371_001.DInput[13]);
	gMachine.In.ProductDetect.pPDCarriageSignalL2 := ADR(X20DIF371_001.DInput[14]);
	//Reserve01.DInput[1]	:= X20DIF371_001.DInput[15];
	//Reserve01.DInput[1]	:= X20DIF371_001.DInput[16];

	// Reset and Mute with the same digital signal
	T_Reset.IN := X20DIF371_001.DInput[12];
	T_Reset.PT := t#250ms;
	T_Reset();

	T_Mute.IN := X20DIF371_001.DInput[12];
	T_Mute.PT := t#100ms;
	T_Mute();

	gMachine.In.Buttons.xReset:= T_Reset.Q;
	gMachine.In.Buttons.xMute:= T_Mute.Q;

	// X20DIF371_002
	gInksInputs[1].xPrintHeadsPsuOK		:= X20DIF371_002.DInput[1];
	gInksInputs[2].xPrintHeadsPsuOK		:= X20DIF371_002.DInput[2];
	gInksInputs[3].xPrintHeadsPsuOK		:= X20DIF371_002.DInput[3];
	gInksInputs[4].xPrintHeadsPsuOK		:= X20DIF371_002.DInput[4];
	gInksInputs[5].xPrintHeadsPsuOK		:= X20DIF371_002.DInput[5];
	gInksInputs[6].xPrintHeadsPsuOK		:= X20DIF371_002.DInput[6];
	gInksInputs[7].xPrintHeadsPsuOK		:= X20DIF371_002.DInput[7];
	gInksInputs[8].xPrintHeadsPsuOK		:= X20DIF371_002.DInput[8];
	gBlockInputs[1].xHeaterDcOkBusBar1	:= X20DIF371_002.DInput[9];
	gBelt.parameters.xDriveProtectionOK	:= X20DIF371_002.DInput[10];
	gBlockInputs[1].xDriveProtectionOK	:= X20DIF371_002.DInput[11];
	gBlockInputs[1].xDifferentialOK		:= X20DIF371_002.DInput[12];
	gMachine.In.x24Vdc					:= X20DIF371_002.DInput[13];
	gBlockInputs[1].Safety.xCurtainEnable01	:= X20DIF371_002.DInput[14];//Same Input
	gBlockInputs[1].Safety.xCurtainEnable02	:= X20DIF371_002.DInput[14];//Same Input
	gBlockInputs[1].Safety.xRearSafetyOK		:= X20DIF371_002.DInput[15];
	gBlockInputs[1].Safety.xSafetyOK			:= X20DIF371_002.DInput[16];

	// X20DIF371_003
	gMachine.In.UPSs[1].xSystemFault			:= NOT X20DIF371_003.DInput[1];
	gMachine.In.UPSs[1].xPowerFault				:= NOT X20DIF371_003.DInput[2];
	gMachine.In.UPSs[1].xLowBattery					:= NOT X20DIF371_003.DInput[3];
	gMachine.In.UPSs[1].xByPass					:= NOT X20DIF371_003.DInput[4];
	gMachine.In.UPSs[2].xSystemFault			:= NOT X20DIF371_003.DInput[5];
	gMachine.In.UPSs[2].xPowerFault				:= NOT X20DIF371_003.DInput[6];
	gMachine.In.UPSs[2].xLowBattery					:= NOT X20DIF371_003.DInput[7];
	gMachine.In.UPSs[2].xByPass					:= NOT X20DIF371_003.DInput[8];
	gBlockInputs[1].xReferenceDI				:= X20DIF371_003.DInput[9];
	//Reserve01.DInput[1]						:= NOT X20DIF371_003.DInput[10];
	gMachine.In.ProductDetect.pPDSignalSensorL1	:= ADR(X20DIF371_003.DInput[11]);
	gMachine.In.ProductDetect.pPDSignalSensorL2	:= ADR(X20DIF371_003.DInput[12]);

//  Those variables are not mapped. Are fast and assigned with pointer
//	gPhotoCells.Inputs.Signals.xPhotoCells[1]		:= X20DIF371_003.DInput[13];//Same Input
	gDing.In.xDingLow							:= X20DIF371_003.DInput[13];//Same Input
//	gPhotoCells.Inputs.Signals.xPhotoCells[2]		:= X20DIF371_003.DInput[14];
//	gPhotoCells.Inputs.Signals.xPhotoCells[3]		:= X20DIF371_003.DInput[15];//Same Input
	gDing.In.xDingHigh							:= X20DIF371_003.DInput[15];//Same Input
	//Reserve01.DInput[1]						:= X20DIF371_003.DInput[16];

	// X20DIF371_004
	gInksInputs[1].xKlixonTriggered		:=X20DIF371_004.DInput[1];
	gInksInputs[2].xKlixonTriggered		:=X20DIF371_004.DInput[2];
	gInksInputs[3].xKlixonTriggered		:=X20DIF371_004.DInput[3];
	gInksInputs[4].xKlixonTriggered		:=X20DIF371_004.DInput[4];
	gInksInputs[5].xKlixonTriggered		:=X20DIF371_004.DInput[5];
	gInksInputs[6].xKlixonTriggered		:=X20DIF371_004.DInput[6];
	gInksInputs[7].xKlixonTriggered		:=X20DIF371_004.DInput[7];
	gInksInputs[8].xKlixonTriggered		:=X20DIF371_004.DInput[8];
	gInksInputs[1].xMinLevel			:=X20DIF371_004.DInput[9];
	gInksInputs[2].xMinLevel			:=X20DIF371_004.DInput[10];
	gInksInputs[3].xMinLevel			:=X20DIF371_004.DInput[11];
	gInksInputs[4].xMinLevel			:=X20DIF371_004.DInput[12];
	gInksInputs[5].xMinLevel			:=X20DIF371_004.DInput[13];
	gInksInputs[6].xMinLevel			:=X20DIF371_004.DInput[14];
	gInksInputs[7].xMinLevel			:=X20DIF371_004.DInput[15];
	gInksInputs[8].xMinLevel			:=X20DIF371_004.DInput[16];

	// X20DIF371_005
	gInksInputs[1].xMaxLevel		:= X20DIF371_005.DInput[1];
	gInksInputs[2].xMaxLevel		:= X20DIF371_005.DInput[2];
	gInksInputs[3].xMaxLevel		:= X20DIF371_005.DInput[3];
	gInksInputs[4].xMaxLevel		:= X20DIF371_005.DInput[4];
	gInksInputs[5].xMaxLevel		:= X20DIF371_005.DInput[5];
	gInksInputs[6].xMaxLevel		:= X20DIF371_005.DInput[6];
	gInksInputs[7].xMaxLevel		:= X20DIF371_005.DInput[7];
	gInksInputs[8].xMaxLevel		:= X20DIF371_005.DInput[8];
	gInksInputs[1].xOverpressure	:= NOT X20DIF371_005.DInput[9];
	gInksInputs[2].xOverpressure 	:= NOT X20DIF371_005.DInput[10];
	gInksInputs[3].xOverpressure 	:= NOT X20DIF371_005.DInput[11];
	gInksInputs[4].xOverpressure	:= NOT X20DIF371_005.DInput[12];
	gInksInputs[5].xOverpressure 	:= NOT X20DIF371_005.DInput[13];
	gInksInputs[6].xOverpressure 	:= NOT X20DIF371_005.DInput[14];
	gInksInputs[7].xOverpressure 	:= NOT X20DIF371_005.DInput[15];
	gInksInputs[8].xOverpressure 	:= NOT X20DIF371_005.DInput[16];

	// X20DIF371_006
	gMachine.In.xPbfCardOK 				:= X20DIF371_006.ModuleOk;
	gMachine.In.iRelieve1.0				:= X20DIF371_006.DInput[1];
	gMachine.In.iRelieve1.1				:= X20DIF371_006.DInput[2];
	gMachine.In.iRelieve1.2				:= X20DIF371_006.DInput[3];
	gMachine.In.iRelieve1.3				:= X20DIF371_006.DInput[4];
	gMachine.In.iRelieve1.4				:= X20DIF371_006.DInput[5];
	gMachine.In.iRelieve1.5				:= X20DIF371_006.DInput[6];
	gMachine.In.iRelieve1.6				:= X20DIF371_006.DInput[7];
	gMachine.In.iRelieve1.7				:= X20DIF371_006.DInput[8];
	gMachine.In.iRelieve1.8				:= X20DIF371_006.DInput[9];
	gMachine.In.xConsentL1Ok			:= X20DIF371_006.DInput[10];
	gMachine.In.xConsentL2Ok			:= X20DIF371_006.DInput[11];
	gMachine.In.xExternalCleaningOrder	:= X20DIF371_006.DInput[12];
	gBlockInputs[1].xWaterLevelSensor	:= X20DIF371_006.DInput[13];
	gBlockInputs[1].xWaterPresureSensor	:= X20DIF371_006.DInput[14];
	//Reserve01.DInput[0]				:= X20DIF371_006.DInput[15];
	//Reserve01.DInput[0]				:= X20DIF371_006.DInput[16];

	// X20DI9372_008
	gBlockInputs[1].xPrintHeadPSU[1]		:= X20DI9372_008.DInput[1];
	gBlockInputs[1].xPrintHeadPSU[2]		:= X20DI9372_008.DInput[2];
	gBlockInputs[1].xPrintHeadPSU[3]		:= X20DI9372_008.DInput[3];
	gBlockInputs[1].xPrintHeadPSU[4]		:= X20DI9372_008.DInput[4];
	gBlockInputs[1].xPrintHeadPSU[5]		:= X20DI9372_008.DInput[5];
	gBlockInputs[1].xPrintHeadPSU[6]		:= X20DI9372_008.DInput[6];
	gBlockInputs[1].xHeaterDcOkPsu[1]	:= X20DI9372_008.DInput[7];
	gBlockInputs[1].xHeaterDcOkPsu[2]	:= X20DI9372_008.DInput[8];
	gBlockInputs[1].xHeaterDcOkPsu[3]	:= X20DI9372_008.DInput[9];
	//Reserve01.DInput[0]			:=X20DI9372_008.DInput[10];
	//Reserve01.DInput[0]			:=X20DI9372_008.DInput[11];
	//Reserve01.DInput[0]			:=X20DI9372_008.DInput[12];

	// X20AI8321_015		(*  BAR A *) (*  BAR B *) (*  BAR C *) (*  BAR D *)
	gInksInputs[1].iVacuum1Raw			:= X20AI8321_015.AInput[1];
	gInksInputs[1].xVacuum1SensorError	:= StatusAnalogInputBroken(X20AI8321_015.ModuleOk, X20AI8321_015.Status01, X20AI8321_015.Status02, 1);
	gInksInputs[1].iVacuum2Raw			:= X20AI8321_015.AInput[2];
	gInksInputs[1].xVacuum2SensorError	:= StatusAnalogInputBroken(X20AI8321_015.ModuleOk, X20AI8321_015.Status01, X20AI8321_015.Status02, 2);
	gInksInputs[2].iVacuum1Raw			:= X20AI8321_015.AInput[3];
	gInksInputs[2].xVacuum1SensorError	:= StatusAnalogInputBroken(X20AI8321_015.ModuleOk, X20AI8321_015.Status01, X20AI8321_015.Status02, 3);
	gInksInputs[2].iVacuum2Raw			:= X20AI8321_015.AInput[4];
	gInksInputs[2].xVacuum2SensorError	:= StatusAnalogInputBroken(X20AI8321_015.ModuleOk, X20AI8321_015.Status01, X20AI8321_015.Status02, 4);
	gInksInputs[3].iVacuum1Raw			:= X20AI8321_015.AInput[5];
	gInksInputs[3].xVacuum1SensorError	:= StatusAnalogInputBroken(X20AI8321_015.ModuleOk, X20AI8321_015.Status01, X20AI8321_015.Status02, 5);
	gInksInputs[3].iVacuum2Raw			:= X20AI8321_015.AInput[6];
	gInksInputs[3].xVacuum2SensorError	:= StatusAnalogInputBroken(X20AI8321_015.ModuleOk, X20AI8321_015.Status01, X20AI8321_015.Status02, 6);
	gInksInputs[4].iVacuum1Raw			:= X20AI8321_015.AInput[7];
	gInksInputs[4].xVacuum1SensorError	:= StatusAnalogInputBroken(X20AI8321_015.ModuleOk, X20AI8321_015.Status01, X20AI8321_015.Status02, 7);
	gInksInputs[4].iVacuum2Raw			:= X20AI8321_015.AInput[8];
	gInksInputs[4].xVacuum2SensorError	:= StatusAnalogInputBroken(X20AI8321_015.ModuleOk, X20AI8321_015.Status01, X20AI8321_015.Status02, 8);

	// X20AI8321_016		(* BAR E *) (* BAR F *) (* BAR G *) (* BAR H *)
	gInksInputs[5].iVacuum1Raw			:= X20AI8321_016.AInput[1];
	gInksInputs[5].xVacuum1SensorError	:= StatusAnalogInputBroken(X20AI8321_016.ModuleOk, X20AI8321_016.Status01, X20AI8321_016.Status02, 1);
	gInksInputs[5].iVacuum2Raw			:= X20AI8321_016.AInput[2];
	gInksInputs[5].xVacuum2SensorError	:= StatusAnalogInputBroken(X20AI8321_016.ModuleOk, X20AI8321_016.Status01, X20AI8321_016.Status02, 2);
	gInksInputs[6].iVacuum1Raw			:= X20AI8321_016.AInput[3];
	gInksInputs[6].xVacuum1SensorError	:= StatusAnalogInputBroken(X20AI8321_016.ModuleOk, X20AI8321_016.Status01, X20AI8321_016.Status02, 3);
	gInksInputs[6].iVacuum2Raw			:= X20AI8321_016.AInput[4];
	gInksInputs[6].xVacuum2SensorError	:= StatusAnalogInputBroken(X20AI8321_016.ModuleOk, X20AI8321_016.Status01, X20AI8321_016.Status02, 4);
	gInksInputs[7].iVacuum1Raw			:= X20AI8321_016.AInput[5];
	gInksInputs[7].xVacuum1SensorError	:= StatusAnalogInputBroken(X20AI8321_016.ModuleOk, X20AI8321_016.Status01, X20AI8321_016.Status02, 5);
	gInksInputs[7].iVacuum2Raw			:= X20AI8321_016.AInput[6];
	gInksInputs[7].xVacuum2SensorError	:= StatusAnalogInputBroken(X20AI8321_016.ModuleOk, X20AI8321_016.Status01, X20AI8321_016.Status02, 6);
	gInksInputs[8].iVacuum1Raw			:= X20AI8321_016.AInput[7];
	gInksInputs[8].xVacuum1SensorError	:= StatusAnalogInputBroken(X20AI8321_016.ModuleOk, X20AI8321_016.Status01, X20AI8321_016.Status02, 7);
	gInksInputs[8].iVacuum2Raw			:= X20AI8321_016.AInput[8];
	gInksInputs[8].xVacuum2SensorError	:= StatusAnalogInputBroken(X20AI8321_016.ModuleOk, X20AI8321_016.Status01, X20AI8321_016.Status02, 8);

	// X20AT4222_22
	gBlockInputs[1].xModuleTemp01Ok		:= X20AT4222_022.ModuleOk;
	gInksInputs[1].iTemperatureRaw		:= X20AT4222_022.TempInput[1];
	gInksInputs[1].xTempSensorError		:= StatusTemperatureInput(X20AT4222_022.Status01, 1);
	gInksInputs[2].iTemperatureRaw		:= X20AT4222_022.TempInput[2];
	gInksInputs[2].xTempSensorError		:= StatusTemperatureInput(X20AT4222_022.Status01, 2);
	gInksInputs[3].iTemperatureRaw		:= X20AT4222_022.TempInput[3];
	gInksInputs[3].xTempSensorError		:= StatusTemperatureInput(X20AT4222_022.Status01, 3);
	gInksInputs[4].iTemperatureRaw		:= X20AT4222_022.TempInput[4];
	gInksInputs[4].xTempSensorError		:= StatusTemperatureInput(X20AT4222_022.Status01, 4);

	// X20AT4222_23
	gBlockInputs[1].xModuleTemp02Ok		:= X20AT4222_023.ModuleOk;
	gInksInputs[5].iTemperatureRaw		:= X20AT4222_023.TempInput[1];
	gInksInputs[5].xTempSensorError		:= StatusTemperatureInput(X20AT4222_023.Status01, 1);
	gInksInputs[6].iTemperatureRaw		:= X20AT4222_023.TempInput[2];
	gInksInputs[6].xTempSensorError		:= StatusTemperatureInput(X20AT4222_023.Status01, 2);
	gInksInputs[7].iTemperatureRaw		:= X20AT4222_023.TempInput[3];
	gInksInputs[7].xTempSensorError		:= StatusTemperatureInput(X20AT4222_023.Status01, 3);
	gInksInputs[8].iTemperatureRaw		:= X20AT4222_023.TempInput[4];
	gInksInputs[8].xTempSensorError		:= StatusTemperatureInput(X20AT4222_023.Status01, 4);

	//X20DIF371_024
	gJamInputs[1].xJamCrash[1]			:= X20DIF371_024.DInput[1];
	gJamInputs[1].xJamCrash[2]			:= X20DIF371_024.DInput[2];
	gJamInputs[1].xJamCrash[3]			:= X20DIF371_024.DInput[3];
	gJamInputs[1].xJamCrash[4]			:= X20DIF371_024.DInput[4];
	gJamInputs[2].xJamCrash[1]			:= X20DIF371_024.DInput[5];
	gJamInputs[2].xJamCrash[2]			:= X20DIF371_024.DInput[6];
	gJamInputs[2].xJamCrash[3]			:= X20DIF371_024.DInput[7];
	gJamInputs[2].xJamCrash[4]			:= X20DIF371_024.DInput[8];
	//JamDetection Crash N1				:= X20DIF371_024.DInput[9];  Not Used
	//JamDetection Crash N2				:= X20DIF371_024.DInput[10]; Not Used
	gJamInputs[1].xJamTestOk			:= X20DIF371_024.DInput[11];
	gJamInputs[2].xJamTestOk			:= X20DIF371_024.DInput[12];
	gTransVacuum[1].Inputs.xBlowersAnyCB	:= NOT X20DIF371_024.DInput[13];
	gNonCrash[1].Inputs.xDiffContacOk	:= X20DIF371_024.DInput[14];
	//Reserve01.DInput[0]				:= X20DIF371_024.DInput[15];
	//Reserve01.DInput[0]				:= X20DIF371_024.DInput[16];

	//X20AI8321_025
	gTransVacuum[2].Inputs.iPressureRaw	:= X20AI8321_025.AInput[1];
	gTransVacuum[2].Inputs.xPressureSensorError	:= StatusAnalogInputBroken(X20AI8321_025.ModuleOk, X20AI8321_025.Status01, X20AI8321_025.Status02, 1);
	gTransVacuum[1].Inputs.iPressureRaw	:= X20AI8321_025.AInput[2];
	gTransVacuum[1].Inputs.xPressureSensorError	:= StatusAnalogInputBroken(X20AI8321_025.ModuleOk, X20AI8321_025.Status01, X20AI8321_025.Status02, 2);

	//NOTE: This code is in IN_Thickness program, to be sure to have it ready prior to work with it

	// X20AI2636_100
	gDing.In.xModuleOK := X20AI2636_100.ModuleOk;
	gDing.In.xDingChannelFault := X20AI2636_100.DInput[1];

	gTransVacuum[2].Inputs.xBlowersAnyCB := gTransVacuum[1].Inputs.xBlowersAnyCB;

	// X20AT4222_029
	gBlockInputs[1].xModuleTemp03Ok		:= X20AT4222_029.ModuleOk;
	gInksInputs[1].iTemperatureTankRaw	:= X20AT4222_029.TempInput[1];
	gInksInputs[1].xTempTankSensorError	:= StatusTemperatureInput(X20AT4222_029.Status01, 1);
	gInksInputs[2].iTemperatureTankRaw	:= X20AT4222_029.TempInput[2];
	gInksInputs[2].xTempTankSensorError	:= StatusTemperatureInput(X20AT4222_029.Status01, 2);
	gInksInputs[3].iTemperatureTankRaw	:= X20AT4222_029.TempInput[3];
	gInksInputs[3].xTempTankSensorError	:= StatusTemperatureInput(X20AT4222_029.Status01, 3);
	gInksInputs[4].iTemperatureTankRaw	:= X20AT4222_029.TempInput[4];
	gInksInputs[4].xTempTankSensorError	:= StatusTemperatureInput(X20AT4222_029.Status01, 4);

	// X20AT4222_030
	gBlockInputs[1].xModuleTemp04Ok		:= X20AT4222_030.ModuleOk;
	gInksInputs[5].iTemperatureTankRaw	:= X20AT4222_030.TempInput[1];
	gInksInputs[5].xTempTankSensorError	:= StatusTemperatureInput(X20AT4222_030.Status01, 1);
	gInksInputs[6].iTemperatureTankRaw	:= X20AT4222_030.TempInput[2];
	gInksInputs[6].xTempTankSensorError	:= StatusTemperatureInput(X20AT4222_030.Status01, 2);
	gInksInputs[7].iTemperatureTankRaw	:= X20AT4222_030.TempInput[3];
	gInksInputs[7].xTempTankSensorError	:= StatusTemperatureInput(X20AT4222_030.Status01, 3);
	gInksInputs[8].iTemperatureTankRaw	:= X20AT4222_030.TempInput[4];
	gInksInputs[8].xTempTankSensorError	:= StatusTemperatureInput(X20AT4222_030.Status01, 4);

	// SI UNIT BK1
	gBlockInputs[1].xSiUnitModuleOk		:= SiUnitPwrLnkBK1.ModuleOk;
	gMachine.In.xAirSupply				:= SiUnitPwrLnkBK1.Input01_16.0;
	gBlockInputs[1].xAirVenturiOK		:= SiUnitPwrLnkBK1.Input01_16.1;
	gBlockInputs[1].xTrayOut			:= SiUnitPwrLnkBK1.Input01_16.2;
	gBlockInputs[1].xIclaSensor			:= SiUnitPwrLnkBK1.Input01_16.3;
	gTransVacuum[1].Inputs.xVaccAirFlow	:= SiUnitPwrLnkBK1.Input01_16.4;
	gTransVacuum[1].Inputs.xJointSystemPressure:= SiUnitPwrLnkBK1.Input01_16.5;
	gBlockInputs[1].xBarsIn := TRUE;
	gTransVacuum[1].Inputs.xSafetyEnable := gTransVacuum[2].Inputs.xSafetyEnable := TRUE; //gMachine.In.xSafetyEnabled;

	gTransVacuum[2].Inputs.xJointSystemPressure := gTransVacuum[1].Inputs.xJointSystemPressure; //Repeat inputs
	gTransVacuum[2].Inputs.xVaccAirFlow	:= gTransVacuum[1].Inputs.xVaccAirFlow;

	//Signals Forced by Configuration
	gBlockInputs[1].Safety.xFrontSafetyOK	:= TRUE;
	gBlockInputs[2].Safety.xFrontSafetyOK	:= TRUE;

	gBlockInputs[1].Safety.xFrontEStopOK := TRUE;
	gBlockInputs[2].Safety.xFrontEStopOK := TRUE;

	gBlockInputs[1].Safety.xRearEStopOK := TRUE;
	gBlockInputs[2].Safety.xRearEStopOK := TRUE;

	gAxisInverter[1].ElecSignals.In.xBreakerOK := TRUE;
	gAxisInverter[2].ElecSignals.In.xBreakerOK := TRUE;
	gAxisInverter[3].ElecSignals.In.xBreakerOK := TRUE;
	gAxisInverter[4].ElecSignals.In.xBreakerOK := TRUE;
	gAxisInverter[5].ElecSignals.In.xBreakerOK := TRUE;
	gAxisInverter[6].ElecSignals.In.xBreakerOK := TRUE;

	//////////////////////////////////\\\\\\\\\\\\\\\\\\\\\\\\\\\\

	// TODO:
	// - Revisar las señales forzadas de esta máquina

	FOR iIndexBlock := 1 TO gMachine.Pt.CT.iNumBlocks DO

		gBlockInputs[iIndexBlock].xHeaterDcOkBusBar2 := TRUE;
		gBlockInputs[iIndexBlock].xHeaterAcOkPsu[1] := TRUE;
		gBlockInputs[iIndexBlock].xHeaterAcOkPsu[2] := TRUE;
		gBlockInputs[iIndexBlock].xHeaterAcOkPsu[3] := TRUE;

		gBlock[iIndexBlock].parameters.Hw.iNumPrintheadsPSU := 6;
		gBlock[iIndexBlock].parameters.Hw.iNumHeaterPSU := 3;

	END_FOR

END_ACTION
```

#### InputsP5.st - PhysicalInputs
```iecst
ACTION InputsP5:

(* CABINET 01 *)

	// X20DIF371_001

	// gMachine.In.iMachineModelCode assigned in an specific Action

	gMachine.In.Buttons.xStart			:= X20DIF371_001.DInput[7];
	gMachine.In.Buttons.xStop			:= NOT X20DIF371_001.DInput[8];
	gMachine.In.Buttons.xAuto			:= X20DIF371_001.DInput[9];
	gMachine.In.Buttons.xZero			:= NOT X20DIF371_001.DInput[10];
	gMachine.In.Buttons.xManual			:= X20DIF371_001.DInput[11];
	//gMachine.In.Buttons.xReset		:= X20DIF371_001.DInput[12];
	gMachine.In.ProductDetect.pPDCarriageSignalL1 := ADR(X20DIF371_001.DInput[13]);
	gMachine.In.ProductDetect.pPDCarriageSignalL2 := ADR(X20DIF371_001.DInput[14]);
	//Reserve01.DInput[1]			:= X20DIF371_001.DInput[15];
	//Reserve01.DInput[1]	:= X20DIF371_001.DInput[16];

	// Reset and Mute with the same digital signal
	T_Reset.IN := X20DIF371_001.DInput[12];
	T_Reset.PT := t#250ms;
	T_Reset();

	T_Mute.IN := X20DIF371_001.DInput[12];
	T_Mute.PT := t#100ms;
	T_Mute();

	gMachine.In.Buttons.xReset:= T_Reset.Q;
	gMachine.In.Buttons.xMute:= T_Mute.Q;

	// X20DIF371_002
	gInksInputs[1].xPrintHeadsPsuOK		:= X20DIF371_002.DInput[1];
	gInksInputs[2].xPrintHeadsPsuOK		:= X20DIF371_002.DInput[2];
	gInksInputs[3].xPrintHeadsPsuOK		:= X20DIF371_002.DInput[3];
	gInksInputs[4].xPrintHeadsPsuOK		:= X20DIF371_002.DInput[4];
	gInksInputs[5].xPrintHeadsPsuOK		:= X20DIF371_002.DInput[5];
	gInksInputs[6].xPrintHeadsPsuOK		:= X20DIF371_002.DInput[6];
	gInksInputs[7].xPrintHeadsPsuOK		:= X20DIF371_002.DInput[7];
	gInksInputs[8].xPrintHeadsPsuOK		:= X20DIF371_002.DInput[8];
	gBlockInputs[1].xHeaterDcOkBusBar1	:= X20DIF371_002.DInput[9];
	gBelt.parameters.xDriveProtectionOK	:= X20DIF371_002.DInput[10];
	gBlockInputs[1].xDriveProtectionOK	:= X20DIF371_002.DInput[11];
	gBlockInputs[1].xDifferentialOK		:= X20DIF371_002.DInput[12];
	gMachine.In.x24Vdc					:= X20DIF371_002.DInput[13];
	gBlockInputs[1].Safety.xCurtainEnable01	:= X20DIF371_002.DInput[14];//Same Input
	gBlockInputs[1].Safety.xCurtainEnable02	:= X20DIF371_002.DInput[14];//Same Input
	gBlockInputs[1].Safety.xRearSafetyOK	:= X20DIF371_002.DInput[15];
	gBlockInputs[1].Safety.xSafetyOK			:= X20DIF371_002.DInput[16];

	// X20DIF371_003
	gMachine.In.UPSs[1].xSystemFault			:= NOT X20DIF371_003.DInput[1];
	gMachine.In.UPSs[1].xPowerFault				:= NOT X20DIF371_003.DInput[2];
	gMachine.In.UPSs[1].xLowBattery					:= NOT X20DIF371_003.DInput[3];
	gMachine.In.UPSs[1].xByPass					:= NOT X20DIF371_003.DInput[4];
	gMachine.In.UPSs[2].xSystemFault			:= NOT X20DIF371_003.DInput[5];
	gMachine.In.UPSs[2].xPowerFault				:= NOT X20DIF371_003.DInput[6];
	gMachine.In.UPSs[2].xLowBattery					:= NOT X20DIF371_003.DInput[7];
	gMachine.In.UPSs[2].xByPass					:= NOT X20DIF371_003.DInput[8];
	gBlockInputs[1].xReferenceDI				:= X20DIF371_003.DInput[9];
	gMachine.In.ProductDetect.pPDSignalSensorL1	:= ADR(X20DIF371_003.DInput[11]);
	gMachine.In.ProductDetect.pPDSignalSensorL2	:= ADR(X20DIF371_003.DInput[12]);

	// Those variables are not mapped. Are fast and assigned with pointer
	//gPhotoCells.Inputs.Signals.xPhotoCells[1]		:= NOT X20DIF371_003.DInput[13];//Same Input
	gDing.In.xDingLow							:= X20DIF371_003.DInput[13];//Same Input
	//gPhotoCells.Inputs.Signals.xPhotoCells[2]		:= NOT X20DIF371_003.DInput[14];
	//gPhotoCells.Inputs.Signals.xPhotoCells[3]		:= NOT X20DIF371_003.DInput[15];//Same Input
	gDing.In.xDingHigh							:= X20DIF371_003.DInput[15];//Same Input
	//Reserve01.DInput[1]						:= X20DIF371_003.DInput[16];

	// X20DIF371_004
	gInksInputs[1].xKlixonTriggered		:=X20DIF371_004.DInput[1];
	gInksInputs[2].xKlixonTriggered		:=X20DIF371_004.DInput[2];
	gInksInputs[3].xKlixonTriggered		:=X20DIF371_004.DInput[3];
	gInksInputs[4].xKlixonTriggered		:=X20DIF371_004.DInput[4];
	gInksInputs[5].xKlixonTriggered		:=X20DIF371_004.DInput[5];
	gInksInputs[6].xKlixonTriggered		:=X20DIF371_004.DInput[6];
	gInksInputs[7].xKlixonTriggered		:=X20DIF371_004.DInput[7];
	gInksInputs[8].xKlixonTriggered		:=X20DIF371_004.DInput[8];
	gInksInputs[1].xMinLevel			:=X20DIF371_004.DInput[9];
	gInksInputs[2].xMinLevel			:=X20DIF371_004.DInput[10];
	gInksInputs[3].xMinLevel			:=X20DIF371_004.DInput[11];
	gInksInputs[4].xMinLevel			:=X20DIF371_004.DInput[12];
	gInksInputs[5].xMinLevel			:=X20DIF371_004.DInput[13];
	gInksInputs[6].xMinLevel			:=X20DIF371_004.DInput[14];
	gInksInputs[7].xMinLevel			:=X20DIF371_004.DInput[15];
	gInksInputs[8].xMinLevel			:=X20DIF371_004.DInput[16];

	// X20DIF371_005
	gInksInputs[1].xMaxLevel		:= X20DIF371_005.DInput[1];
	gInksInputs[2].xMaxLevel		:= X20DIF371_005.DInput[2];
	gInksInputs[3].xMaxLevel		:= X20DIF371_005.DInput[3];
	gInksInputs[4].xMaxLevel		:= X20DIF371_005.DInput[4];
	gInksInputs[5].xMaxLevel		:= X20DIF371_005.DInput[5];
	gInksInputs[6].xMaxLevel		:= X20DIF371_005.DInput[6];
	gInksInputs[7].xMaxLevel		:= X20DIF371_005.DInput[7];
	gInksInputs[8].xMaxLevel		:= X20DIF371_005.DInput[8];
	gInksInputs[1].xOverpressure	:= NOT X20DIF371_005.DInput[9];
	gInksInputs[2].xOverpressure 	:= NOT X20DIF371_005.DInput[10];
	gInksInputs[3].xOverpressure 	:= NOT X20DIF371_005.DInput[11];
	gInksInputs[4].xOverpressure	:= NOT X20DIF371_005.DInput[12];
	gInksInputs[5].xOverpressure 	:= NOT X20DIF371_005.DInput[13];
	gInksInputs[6].xOverpressure 	:= NOT X20DIF371_005.DInput[14];
	gInksInputs[7].xOverpressure 	:= NOT X20DIF371_005.DInput[15];
	gInksInputs[8].xOverpressure 	:= NOT X20DIF371_005.DInput[16];

	// X20DIF371_006
	gMachine.In.xPbfCardOK 				:= X20DIF371_006.ModuleOk;
	gMachine.In.iRelieve1.0				:= X20DIF371_006.DInput[1];
	gMachine.In.iRelieve1.1				:= X20DIF371_006.DInput[2];
	gMachine.In.iRelieve1.2				:= X20DIF371_006.DInput[3];
	gMachine.In.iRelieve1.3				:= X20DIF371_006.DInput[4];
	gMachine.In.iRelieve1.4				:= X20DIF371_006.DInput[5];
	gMachine.In.iRelieve1.5				:= X20DIF371_006.DInput[6];
	gMachine.In.iRelieve1.6				:= X20DIF371_006.DInput[7];
	gMachine.In.iRelieve1.7				:= X20DIF371_006.DInput[8];
	gMachine.In.iRelieve1.8				:= X20DIF371_006.DInput[9];
	gMachine.In.xConsentL1Ok			:= X20DIF371_006.DInput[10];
	gMachine.In.xConsentL2Ok			:= X20DIF371_006.DInput[11];
	gMachine.In.xExternalCleaningOrder	:= X20DIF371_006.DInput[12];
	gBlockInputs[1].xWaterLevelSensor	:= X20DIF371_006.DInput[13];
	gBlockInputs[1].xWaterPresureSensor	:= X20DIF371_006.DInput[14];
	//Reserve01.DInput[0]				:= X20DIF371_006.DInput[15];
	//Reserve01.DInput[0]				:= X20DIF371_006.DInput[16];

	// X20DI9372_008
	gBlockInputs[1].xPrintHeadPSU[1]		:= X20DI9372_008.DInput[1];
	gBlockInputs[1].xPrintHeadPSU[2]		:= X20DI9372_008.DInput[2];
	gBlockInputs[1].xPrintHeadPSU[3]		:= X20DI9372_008.DInput[3];
	gBlockInputs[1].xPrintHeadPSU[4]		:= X20DI9372_008.DInput[4];
	gBlockInputs[1].xPrintHeadPSU[5]		:= X20DI9372_008.DInput[5];
	gBlockInputs[1].xPrintHeadPSU[6]		:= X20DI9372_008.DInput[6];
	gBlockInputs[1].xHeaterDcOkPsu[1]	:= X20DI9372_008.DInput[7];
	gBlockInputs[1].xHeaterDcOkPsu[2]	:= X20DI9372_008.DInput[8];
	gBlockInputs[1].xHeaterDcOkPsu[3]	:= X20DI9372_008.DInput[9];
	//Reserve01.DInput[0]			:=X20DI9372_008.DInput[10];
	//Reserve01.DInput[0]			:=X20DI9372_008.DInput[11];
	//Reserve01.DInput[0]			:=X20DI9372_008.DInput[12];

	// X20AI8321_015		(*  BAR A *) (*  BAR B *) (*  BAR C *) (*  BAR D *)
	gInksInputs[1].iVacuum1Raw			:= X20AI8321_015.AInput[1];
	gInksInputs[1].xVacuum1SensorError	:= StatusAnalogInputBroken(X20AI8321_015.ModuleOk, X20AI8321_015.Status01, X20AI8321_015.Status02, 1);
	gInksInputs[1].iVacuum2Raw			:= X20AI8321_015.AInput[2];
	gInksInputs[1].xVacuum2SensorError	:= StatusAnalogInputBroken(X20AI8321_015.ModuleOk, X20AI8321_015.Status01, X20AI8321_015.Status02, 2);
	gInksInputs[2].iVacuum1Raw			:= X20AI8321_015.AInput[3];
	gInksInputs[2].xVacuum1SensorError	:= StatusAnalogInputBroken(X20AI8321_015.ModuleOk, X20AI8321_015.Status01, X20AI8321_015.Status02, 3);
	gInksInputs[2].iVacuum2Raw			:= X20AI8321_015.AInput[4];
	gInksInputs[2].xVacuum2SensorError	:= StatusAnalogInputBroken(X20AI8321_015.ModuleOk, X20AI8321_015.Status01, X20AI8321_015.Status02, 4);
	gInksInputs[3].iVacuum1Raw			:= X20AI8321_015.AInput[5];
	gInksInputs[3].xVacuum1SensorError	:= StatusAnalogInputBroken(X20AI8321_015.ModuleOk, X20AI8321_015.Status01, X20AI8321_015.Status02, 5);
	gInksInputs[3].iVacuum2Raw			:= X20AI8321_015.AInput[6];
	gInksInputs[3].xVacuum2SensorError	:= StatusAnalogInputBroken(X20AI8321_015.ModuleOk, X20AI8321_015.Status01, X20AI8321_015.Status02, 6);
	gInksInputs[4].iVacuum1Raw			:= X20AI8321_015.AInput[7];
	gInksInputs[4].xVacuum1SensorError	:= StatusAnalogInputBroken(X20AI8321_015.ModuleOk, X20AI8321_015.Status01, X20AI8321_015.Status02, 7);
	gInksInputs[4].iVacuum2Raw			:= X20AI8321_015.AInput[8];
	gInksInputs[4].xVacuum2SensorError	:= StatusAnalogInputBroken(X20AI8321_015.ModuleOk, X20AI8321_015.Status01, X20AI8321_015.Status02, 8);

	// X20AI8321_016		(* BAR E *) (* BAR F *) (* BAR G *) (* BAR H *)
	gInksInputs[5].iVacuum1Raw			:= X20AI8321_016.AInput[1];
	gInksInputs[5].xVacuum1SensorError	:= StatusAnalogInputBroken(X20AI8321_016.ModuleOk, X20AI8321_016.Status01, X20AI8321_016.Status02, 1);
	gInksInputs[5].iVacuum2Raw			:= X20AI8321_016.AInput[2];
	gInksInputs[5].xVacuum2SensorError	:= StatusAnalogInputBroken(X20AI8321_016.ModuleOk, X20AI8321_016.Status01, X20AI8321_016.Status02, 2);
	gInksInputs[6].iVacuum1Raw			:= X20AI8321_016.AInput[3];
	gInksInputs[6].xVacuum1SensorError	:= StatusAnalogInputBroken(X20AI8321_016.ModuleOk, X20AI8321_016.Status01, X20AI8321_016.Status02, 3);
	gInksInputs[6].iVacuum2Raw			:= X20AI8321_016.AInput[4];
	gInksInputs[6].xVacuum2SensorError	:= StatusAnalogInputBroken(X20AI8321_016.ModuleOk, X20AI8321_016.Status01, X20AI8321_016.Status02, 4);
	gInksInputs[7].iVacuum1Raw			:= X20AI8321_016.AInput[5];
	gInksInputs[7].xVacuum1SensorError	:= StatusAnalogInputBroken(X20AI8321_016.ModuleOk, X20AI8321_016.Status01, X20AI8321_016.Status02, 5);
	gInksInputs[7].iVacuum2Raw			:= X20AI8321_016.AInput[6];
	gInksInputs[7].xVacuum2SensorError	:= StatusAnalogInputBroken(X20AI8321_016.ModuleOk, X20AI8321_016.Status01, X20AI8321_016.Status02, 6);
	gInksInputs[8].iVacuum1Raw			:= X20AI8321_016.AInput[7];
	gInksInputs[8].xVacuum1SensorError	:= StatusAnalogInputBroken(X20AI8321_016.ModuleOk, X20AI8321_016.Status01, X20AI8321_016.Status02, 7);
	gInksInputs[8].iVacuum2Raw			:= X20AI8321_016.AInput[8];
	gInksInputs[8].xVacuum2SensorError	:= StatusAnalogInputBroken(X20AI8321_016.ModuleOk, X20AI8321_016.Status01, X20AI8321_016.Status02, 8);

	// X20AT4222_22
	gBlockInputs[1].xModuleTemp01Ok		:= X20AT4222_022.ModuleOk;
	gInksInputs[1].iTemperatureRaw		:= X20AT4222_022.TempInput[1];
	gInksInputs[1].xTempSensorError		:= StatusTemperatureInput(X20AT4222_022.Status01, 1);
	gInksInputs[2].iTemperatureRaw		:= X20AT4222_022.TempInput[2];
	gInksInputs[2].xTempSensorError		:= StatusTemperatureInput(X20AT4222_022.Status01, 2);
	gInksInputs[3].iTemperatureRaw		:= X20AT4222_022.TempInput[3];
	gInksInputs[3].xTempSensorError		:= StatusTemperatureInput(X20AT4222_022.Status01, 3);
	gInksInputs[4].iTemperatureRaw		:= X20AT4222_022.TempInput[4];
	gInksInputs[4].xTempSensorError		:= StatusTemperatureInput(X20AT4222_022.Status01, 4);

	// X20AT4222_23
	gBlockInputs[1].xModuleTemp02Ok		:= X20AT4222_023.ModuleOk;
	gInksInputs[5].iTemperatureRaw		:= X20AT4222_023.TempInput[1];
	gInksInputs[5].xTempSensorError		:= StatusTemperatureInput(X20AT4222_023.Status01, 1);
	gInksInputs[6].iTemperatureRaw		:= X20AT4222_023.TempInput[2];
	gInksInputs[6].xTempSensorError		:= StatusTemperatureInput(X20AT4222_023.Status01, 2);
	gInksInputs[7].iTemperatureRaw		:= X20AT4222_023.TempInput[3];
	gInksInputs[7].xTempSensorError		:= StatusTemperatureInput(X20AT4222_023.Status01, 3);
	gInksInputs[8].iTemperatureRaw		:= X20AT4222_023.TempInput[4];
	gInksInputs[8].xTempSensorError		:= StatusTemperatureInput(X20AT4222_023.Status01, 4);

	// X20AI2636_024
	gDing.In.xModuleOK := X20AI2636_100.ModuleOk;
	gDing.In.xDingChannelFault := X20AI2636_100.DInput[1];

	// X20SM1436_024 & X20SM1436_025
	gPhotoCells.status.xBackModuleOk := X20SM1436_111.ModuleOk;
	gPhotoCells.status.xFrontModuleOk := X20SM1436_112.ModuleOk;

	// X20AT4222_027
	gBlockInputs[1].xModuleTemp03Ok		:= X20AT4222_027.ModuleOk;
	gInksInputs[1].iTemperatureTankRaw	:= X20AT4222_027.TempInput[1];
	gInksInputs[1].xTempTankSensorError	:= StatusTemperatureInput(X20AT4222_027.Status01, 1);
	gInksInputs[2].iTemperatureTankRaw	:= X20AT4222_027.TempInput[2];
	gInksInputs[2].xTempTankSensorError	:= StatusTemperatureInput(X20AT4222_027.Status01, 2);
	gInksInputs[3].iTemperatureTankRaw	:= X20AT4222_027.TempInput[3];
	gInksInputs[3].xTempTankSensorError	:= StatusTemperatureInput(X20AT4222_027.Status01, 3);
	gInksInputs[4].iTemperatureTankRaw	:= X20AT4222_027.TempInput[4];
	gInksInputs[4].xTempTankSensorError	:= StatusTemperatureInput(X20AT4222_027.Status01, 4);

	// X20AT4222_028
	gBlockInputs[1].xModuleTemp04Ok		:= X20AT4222_028.ModuleOk;
	gInksInputs[5].iTemperatureTankRaw	:= X20AT4222_028.TempInput[1];
	gInksInputs[5].xTempTankSensorError	:= StatusTemperatureInput(X20AT4222_028.Status01, 1);
	gInksInputs[6].iTemperatureTankRaw	:= X20AT4222_028.TempInput[2];
	gInksInputs[6].xTempTankSensorError	:= StatusTemperatureInput(X20AT4222_028.Status01, 2);
	gInksInputs[7].iTemperatureTankRaw	:= X20AT4222_028.TempInput[3];
	gInksInputs[7].xTempTankSensorError	:= StatusTemperatureInput(X20AT4222_028.Status01, 3);
	gInksInputs[8].iTemperatureTankRaw	:= X20AT4222_028.TempInput[4];
	gInksInputs[8].xTempTankSensorError	:= StatusTemperatureInput(X20AT4222_028.Status01, 4);

	// SI UNIT BK1
	gBlockInputs[1].xSiUnitModuleOk		:= SiUnitPwrLnkBK1.ModuleOk;
	gMachine.In.xAirSupply				:= SiUnitPwrLnkBK1.Input01_16.0;
	gBlockInputs[1].xAirVenturiOK		:= SiUnitPwrLnkBK1.Input01_16.1;
	gBlockInputs[1].xTrayOut			:= SiUnitPwrLnkBK1.Input01_16.2;
	gBlockInputs[1].xIclaSensor			:= SiUnitPwrLnkBK1.Input01_16.3;
	gTransVacuum[1].Inputs.xVaccAirFlow	:= SiUnitPwrLnkBK1.Input01_16.4;
	gTransVacuum[1].Inputs.xJointSystemPressure:= SiUnitPwrLnkBK1.Input01_16.5;
	gBlockInputs[1].xBarsIn := TRUE;
	gTransVacuum[1].Inputs.xSafetyEnable := gTransVacuum[2].Inputs.xSafetyEnable := TRUE; //gMachine.In.xSafetyEnabled;

	gTransVacuum[2].Inputs.xJointSystemPressure := gTransVacuum[1].Inputs.xJointSystemPressure; //Repeat inputs
	gTransVacuum[2].Inputs.xVaccAirFlow	:= gTransVacuum[1].Inputs.xVaccAirFlow;

	//Signals Forced by Configuration
	gBlockInputs[1].Safety.xFrontSafetyOK	:= TRUE;
	gBlockInputs[2].Safety.xFrontSafetyOK	:= TRUE;

	gBlockInputs[1].Safety.xFrontEStopOK := TRUE;
	gBlockInputs[2].Safety.xFrontEStopOK := TRUE;

	FOR iIndexBlock := 1 TO gMachine.Pt.CT.iNumBlocks DO

		gBlockInputs[iIndexBlock].xHeaterDcOkBusBar2 := TRUE;
		gBlockInputs[iIndexBlock].xHeaterAcOkPsu[1] := TRUE;
		gBlockInputs[iIndexBlock].xHeaterAcOkPsu[2] := TRUE;
		gBlockInputs[iIndexBlock].xHeaterAcOkPsu[3] := TRUE;

		gBlock[iIndexBlock].parameters.Hw.iNumPrintheadsPSU := 6;
		gBlock[iIndexBlock].parameters.Hw.iNumHeaterPSU := 3;

	END_FOR

END_ACTION
```

#### InputsCube.st - PhysicalInputs
```iecst
ACTION InputsCube:

	//These signals must come from X5?
	gMachine.In.xConsentL1Ok := gSafetyController.Outputs.xPrinterToX5;
	gMachine.In.xConsentL2Ok := gSafetyController.Outputs.xPrinterToX5;

	gCuringLed[iIndexColorCuringLedBar].Signals.Inputs.xFrontDoorClosed := gSafetyController.Inputs.xPrinterFrontDoorSwitch;

	//////////
	//PDC
	//////////
	//PDC X20DIF371_002
	//These inputs are read in MachineConfigurator>InputsMachineModel
	//	:= Pdc_X20DIF371_002.DInput[1];
	//	:= Pdc_X20DIF371_002.DInput[2];
	//	:= Pdc_X20DIF371_002.DInput[3];
	//	:= Pdc_X20DIF371_002.DInput[4];
	//	:= Pdc_X20DIF371_002.DInput[5];
	//	:= Pdc_X20DIF371_002.DInput[6];
	gAxisInverter[1].ElecSignals.In.xBreakerOK	:= Pdc_X20DIF371_002.DInput[7];
	gAxisInverter[2].ElecSignals.In.xBreakerOK	:= Pdc_X20DIF371_002.DInput[8];
	gMachine.In.xOvervoltage  := NOT Pdc_X20DIF371_002.DInput[9];
	//24vdc psu IDS Power alarm	:= Pdc_X20DIF371_002.DInput[10];
	gMachine.In.x24Vdc	:= Pdc_X20DIF371_002.DInput[11];
	//Printer maniobra power supply OK	:= Pdc_X20DIF371_002.DInput[12];
	gMachine.In.xPowerSwitch	:= Pdc_X20DIF371_002.DInput[13];
	gMachine.In.xSafetyEnabled	:= Pdc_X20DIF371_002.DInput[14]; //Enable printer coming direct from safety controller
	// := NOT Pdc_X20DIF371_002.DInput[15];
	// := NOT Pdc_X20DIF371_002.DInput[16];

	//PDC X20DIF371_003
	//Reserved for Ultra(¿?)
	//X5 - 3ph power supply OK := Pdc_X20DIF371_003.DInput[1];
	//X5 - 1ph+n power supply OK	:= Pdc_X20DIF371_003.DInput[2];
	gMachine.In.xRemoteReset	:= Pdc_X20DIF371_003.DInput[3];
	gMachine.In.xRemoteJog	:= Pdc_X20DIF371_003.DInput[4];
	//X5 - MI1	:= Pdc_X20DIF371_003.DInput[5];
	//X5 - MI2	:= Pdc_X20DIF371_003.DInput[6];
	//X5 - MI3	:= Pdc_X20DIF371_003.DInput[7];
	//SPARE	:= Pdc_X20DIF371_003.DInput[8];  ////////// Here goes the CheckMedia signal
	//SPARE	:= Pdc_X20DIF371_003.DInput[9];
	//SPARE	:= Pdc_X20DIF371_003.DInput[10];
	//SPARE := Pdc_X20DIF371_003.DInput[11];
	//SPARE := Pdc_X20DIF371_003.DInput[12];
	//SPARE := Pdc_X20DIF371_003.DInput[13];
	//SPARE := Pdc_X20DIF371_003.DInput[14];

	//PDC X20DIF371_004
	gInksInputs[1].xPrintHeadsPsuOK := Pdc_X20DIF371_004.DInput[1];
	gInksInputs[2].xPrintHeadsPsuOK := Pdc_X20DIF371_004.DInput[2];
	gInksInputs[3].xPrintHeadsPsuOK := Pdc_X20DIF371_004.DInput[3];
	gInksInputs[4].xPrintHeadsPsuOK := Pdc_X20DIF371_004.DInput[4];
	gInksInputs[5].xPrintHeadsPsuOK := Pdc_X20DIF371_004.DInput[5];
	gChiller[gCuringLed[iIndexColorCuringLedBar].Parameters.iChillerIndex].In.xPowered := Pdc_X20DIF371_004.DInput[6];
	gChiller[gCuringLed[iIndexColorCuringLedBar].Parameters.iChillerIndex].In.xCooling := Pdc_X20DIF371_004.DInput[6] AND gChiller[gCuringLed[iIndexColorCuringLedBar].Parameters.iChillerIndex].Out.xStart;
	gChiller[gCuringLed[iIndexColorCuringLedBar].Parameters.iChillerIndex].In.xAlarm := NOT Pdc_X20DIF371_004.DInput[7];

	//PDC X20DIF371_030
	gCuringLed[iIndexColorCuringLedBar].Signals.Inputs.xPsuDcOk[1] := Pdc_X20DIF371_030.DInput[1];
	gCuringLed[iIndexColorCuringLedBar].Signals.Inputs.xPsuAcOk[1] := Pdc_X20DIF371_030.DInput[2];
	gCuringLed[iIndexColorCuringLedBar].Signals.Inputs.xPsuDcOk[2] := Pdc_X20DIF371_030.DInput[3];
	gCuringLed[iIndexColorCuringLedBar].Signals.Inputs.xPsuAcOk[2] := Pdc_X20DIF371_030.DInput[4];
	gCuringLed[iIndexColorCuringLedBar].Signals.Inputs.xPsuDcOk[3] := Pdc_X20DIF371_030.DInput[5];
	gCuringLed[iIndexColorCuringLedBar].Signals.Inputs.xPsuAcOk[3] := Pdc_X20DIF371_030.DInput[6];
	gCuringLed[iIndexColorCuringLedBar].Signals.Inputs.xPsuDcOk[4] := Pdc_X20DIF371_030.DInput[7];
	gCuringLed[iIndexColorCuringLedBar].Signals.Inputs.xPsuAcOk[4] := Pdc_X20DIF371_030.DInput[8];
	gCuringLed[iIndexColorCuringLedBar].Signals.Inputs.xSafetyEnable := gMachine.In.xSafetyEnabled; // NOTE: Check the order of assignation. This one after the machine one
	gBlockInputs[1].xPrintHeadPSU[1] := Pdc_X20DIF371_030.DInput[9] (*DcOk*) AND Pdc_X20DIF371_030.DInput[10] (*DcOk*);
	gBlockInputs[1].xHeaterDcOkPsu[1] := Pdc_X20DIF371_030.DInput[11];
	gBlockInputs[1].xHeaterAcOkPsu[1] := Pdc_X20DIF371_030.DInput[12];

	//PDC X20DIF371_060
	gMachine.In.UPSs[1].LoadOnUtility := Pdc_X20DIF371_060.DInput[1];
	gMachine.In.UPSs[1].LoadOnBattery 	:= gMachine.In.UPSs[1].xPowerFault := Pdc_X20DIF371_060.DInput[2];
	gMachine.In.UPSs[1].xLowBattery 	:= Pdc_X20DIF371_060.DInput[3];
	gMachine.In.UPSs[1].xByPass 		:= Pdc_X20DIF371_060.DInput[4];
	// := Pdc_X20DIF371_030.DInput[5];
	// := Pdc_X20DIF371_030.DInput[6];
	gMachine.In.UPSs[2].LoadOnUtility	:= Pdc_X20DIF371_060.DInput[7];
	gMachine.In.UPSs[2].LoadOnBattery 	:= gMachine.In.UPSs[2].xPowerFault := Pdc_X20DIF371_060.DInput[8];
	gMachine.In.UPSs[2].xLowBattery 	:= Pdc_X20DIF371_060.DInput[9];
	gMachine.In.UPSs[2].xByPass 		:= Pdc_X20DIF371_060.DInput[10];

	//PDC X20DIF371_060
	gAxisInverter[3].ElecSignals.In.xBreakerOK := Pdc_X20DIF371_070.DInput[1];

	//////////
	//PRINTER
	//////////

	//101
	gMachine.In.Buttons.xAuto := X20DIF371_101.DInput[1];
	gMachine.In.Buttons.xZero := NOT X20DIF371_101.DInput[2];
	gMachine.In.Buttons.xManual := X20DIF371_101.DInput[3];
	gMachine.In.Buttons.xReset := X20DIF371_101.DInput[4];

	gMachine.In.ProductDetect.pPDCarriageSignalL1 := ADR(X20DIF371_101.DInput[5]);
	gMachine.In.ProductDetect.pPDCarriageSignalL2	:= ADR(FakeBoolInput);
	gBlockInputs[1].xReferenceDI := X20DIF371_101.DInput[6];
	gMachine.In.ProductDetect.pPDSignalSensorL1	:= ADR(X20DIF371_101.DInput[7]);
	gMachine.In.ProductDetect.pPDSignalSensorL2	:= ADR(FakeBoolInput);
	gDing.In.xDingLow:= X20DIF371_101.DInput[8];
	gDing.In.xDingHigh:= X20DIF371_101.DInput[9];
	gThicknessCtrl.Inputs.CheckMedia[1].xCheckFail := X20DIF371_101.DInput[11] OR NOT Pdc_X20DIF371_003.DInput[8];
	gDing.In.xModuleOK := Pdc_X20AI2636_050.ModuleOk;
	gDing.In.xDingChannelFault := Pdc_X20AI2636_050.DInput[1];

	//102
	gJamInputs[1].xJamCrash[1] := X20DIF371_102.DInput[1];
	gJamInputs[1].xJamCrash[2] := X20DIF371_102.DInput[2];
	gJamInputs[1].xJamCrash[3] := X20DIF371_102.DInput[3];
	gJamInputs[1].xJamCrash[4] := X20DIF371_102.DInput[4];
	gJamInputs[2].xJamCrash[1] := X20DIF371_102.DInput[5];
	gJamInputs[2].xJamCrash[2] := X20DIF371_102.DInput[6];
	gJamInputs[2].xJamCrash[3] := X20DIF371_102.DInput[7];
	gJamInputs[1].xJamLowCrash := X20DIF371_102.DInput[8];
	gJamInputs[1].xJamTestOk := X20DIF371_102.DInput[9];
	gJamInputs[2].xJamLowCrash := X20DIF371_102.DInput[10];
	gJamInputs[2].xJamTestOk := X20DIF371_102.DInput[11];

	//103
	gInksInputs[1].xOverpressure  := NOT X20DIF371_103.DInput[1];
	gInksInputs[2].xOverpressure  := NOT X20DIF371_103.DInput[2];
	gInksInputs[3].xOverpressure  := NOT X20DIF371_103.DInput[3];
	gInksInputs[4].xOverpressure  := NOT X20DIF371_103.DInput[4];
	gInksInputs[5].xOverpressure  := NOT X20DIF371_103.DInput[5];
	//  := X20DIF371_103.DInput[6];
	//  := X20DIF371_103.DInput[7];
	//  := X20DIF371_103.DInput[8];
	// := X20DIF371_103.DInput[9];
	// := X20DIF371_105.DInput[10];
	gInksInputs[1].xKlixonTriggered := NOT X20DIF371_103.DInput[11];
	gInksInputs[2].xKlixonTriggered := NOT X20DIF371_103.DInput[12];
	gInksInputs[3].xKlixonTriggered := NOT X20DIF371_103.DInput[13];
	gInksInputs[4].xKlixonTriggered := NOT X20DIF371_103.DInput[14];
	gInksInputs[5].xKlixonTriggered := NOT X20DIF371_103.DInput[15];

	//104
	//UV Curing leds related
	gCuringLed[iIndexColorCuringLedBar].Lamp[1].Inputs.ThermalFault	:= NOT X20DIF371_104.DInput[1];
	gCuringLed[iIndexColorCuringLedBar].Lamp[1].Inputs.SLMFault		:= NOT X20DIF371_104.DInput[2];
	gCuringLed[iIndexColorCuringLedBar].Lamp[2].Inputs.ThermalFault	:= NOT X20DIF371_104.DInput[3];
	gCuringLed[iIndexColorCuringLedBar].Lamp[2].Inputs.SLMFault		:= NOT X20DIF371_104.DInput[4];
	gCuringLed[iIndexColorCuringLedBar].Lamp[3].Inputs.ThermalFault	:= NOT X20DIF371_104.DInput[5];
	gCuringLed[iIndexColorCuringLedBar].Lamp[3].Inputs.SLMFault		:= NOT X20DIF371_104.DInput[6];
	gCuringLed[iIndexColorCuringLedBar].Signals.Inputs.xN2LowFlow	:= NOT X20DIF371_104.DInput[7];
	gCuringLed[iIndexColorCuringLedBar].Signals.Inputs.xN2HighFlow	:= NOT X20DIF371_104.DInput[8];

	//Analog inputs
	//X20AI8321_111
	gInksInputs[1].iVacuum1Raw := X20AI8321_111.AInput[1];
	gInksInputs[1].xVacuum1SensorError 	:= StatusAnalogInputBroken( X20AI8321_111.ModuleOk, X20AI8321_111.Status01, X20AI8321_111.Status02, 1);
	gInksInputs[1].iVacuum2Raw := X20AI8321_111.AInput[2];
	gInksInputs[1].xVacuum2SensorError 	:= StatusAnalogInputBroken( X20AI8321_111.ModuleOk, X20AI8321_111.Status01, X20AI8321_111.Status02, 2);
	gInksInputs[2].iVacuum1Raw := X20AI8321_111.AInput[3];
	gInksInputs[2].xVacuum1SensorError 	:= StatusAnalogInputBroken( X20AI8321_111.ModuleOk, X20AI8321_111.Status01, X20AI8321_111.Status02, 3);
	gInksInputs[2].iVacuum2Raw := X20AI8321_111.AInput[4];
	gInksInputs[2].xVacuum2SensorError 	:= StatusAnalogInputBroken( X20AI8321_111.ModuleOk, X20AI8321_111.Status01, X20AI8321_111.Status02, 4);
	gInksInputs[3].iVacuum1Raw := X20AI8321_111.AInput[5];
	gInksInputs[3].xVacuum1SensorError 	:= StatusAnalogInputBroken( X20AI8321_111.ModuleOk, X20AI8321_111.Status01, X20AI8321_111.Status02, 5);
	gInksInputs[3].iVacuum2Raw := X20AI8321_111.AInput[6];
	gInksInputs[3].xVacuum2SensorError 	:= StatusAnalogInputBroken( X20AI8321_111.ModuleOk, X20AI8321_111.Status01, X20AI8321_111.Status02, 6);
	gInksInputs[4].iVacuum1Raw := X20AI8321_111.AInput[7];
	gInksInputs[4].xVacuum1SensorError 	:= StatusAnalogInputBroken( X20AI8321_111.ModuleOk, X20AI8321_111.Status01, X20AI8321_111.Status02, 7);
	gInksInputs[4].iVacuum2Raw := X20AI8321_111.AInput[8];
	gInksInputs[4].xVacuum2SensorError 	:= StatusAnalogInputBroken( X20AI8321_111.ModuleOk, X20AI8321_111.Status01, X20AI8321_111.Status02, 8);

	//X20AI8321_112
	gInksInputs[5].iVacuum1Raw := X20AI8321_112.AInput[1];
	gInksInputs[5].xVacuum1SensorError 	:= StatusAnalogInputBroken( X20AI8321_112.ModuleOk, X20AI8321_112.Status01, X20AI8321_112.Status02, 1);
	gInksInputs[5].iVacuum2Raw := X20AI8321_112.AInput[2];
	gInksInputs[5].xVacuum2SensorError 	:= StatusAnalogInputBroken( X20AI8321_112.ModuleOk, X20AI8321_112.Status01, X20AI8321_112.Status02, 2);
	gBlockInputs[1].iHumidityRaw := X20AI8321_112.AInput[3];
	gBlockInputs[1].xHumiditySensorError 	:= StatusAnalogInputBroken( X20AI8321_112.ModuleOk, X20AI8321_112.Status01, X20AI8321_112.Status02, 3);
	gBlockInputs[1].iTemperatureRaw := X20AI8321_112.AInput[4];
	gBlockInputs[1].xTemperatureSensorError	:= StatusAnalogInputBroken( X20AI8321_112.ModuleOk, X20AI8321_112.Status01, X20AI8321_112.Status02, 4);

	//X20AI8321_113
	gTransVacuum[1].Inputs.iPressureRaw := X20AI8321_113.AInput[1];
	gTransVacuum[1].Inputs.xPressureSensorError := StatusAnalogInputBroken( X20AI8321_113.ModuleOk, X20AI8321_113.Status01, X20AI8321_113.Status02, 1);
	gMachine.In.ProductDetect.iAnalogSignal := X20AI8321_113.AInput[2]; //-2mm = 4mA, 10mm = 20mA
	gMachine.In.ProductDetect.xAnalogSignalError := StatusAnalogInputBroken( X20AI8321_113.ModuleOk, X20AI8321_113.Status01, X20AI8321_113.Status02, 2);

	gInksInputs[1].iInTankLevel := X20AI8321_113.AInput[3];
	gInksInputs[1].xInkLevelTankSensorError := StatusAnalogInputBroken( X20AI8321_113.ModuleOk, X20AI8321_113.Status01, X20AI8321_113.Status02, 3);
	gInksInputs[2].iInTankLevel := X20AI8321_113.AInput[4];
	gInksInputs[2].xInkLevelTankSensorError := StatusAnalogInputBroken( X20AI8321_113.ModuleOk, X20AI8321_113.Status01, X20AI8321_113.Status02, 4);
	gInksInputs[3].iInTankLevel := X20AI8321_113.AInput[5];
	gInksInputs[3].xInkLevelTankSensorError := StatusAnalogInputBroken( X20AI8321_113.ModuleOk, X20AI8321_113.Status01, X20AI8321_113.Status02, 5);
	gInksInputs[4].iInTankLevel := X20AI8321_113.AInput[6];
	gInksInputs[4].xInkLevelTankSensorError := StatusAnalogInputBroken( X20AI8321_113.ModuleOk, X20AI8321_113.Status01, X20AI8321_113.Status02, 6);
	gInksInputs[5].iInTankLevel := X20AI8321_113.AInput[7];
	gInksInputs[5].xInkLevelTankSensorError := StatusAnalogInputBroken( X20AI8321_113.ModuleOk, X20AI8321_113.Status01, X20AI8321_113.Status02, 7);

	//PT100
	gBlockInputs[1].xModuleTemp01Ok	:= X20AT4222_119.ModuleOk;
	gInksInputs[1].iTemperatureRaw := X20AT4222_119.TempInput[1];
	gInksInputs[1].xTempSensorError	:= StatusTemperatureInput(X20AT4222_119.Status01, 1) OR NOT X20AT4222_119.ModuleOk;
	gInksInputs[2].iTemperatureRaw := X20AT4222_119.TempInput[2];
	gInksInputs[2].xTempSensorError	:= StatusTemperatureInput(X20AT4222_119.Status01, 2) OR NOT X20AT4222_119.ModuleOk;
	gInksInputs[3].iTemperatureRaw := X20AT4222_119.TempInput[3];
	gInksInputs[3].xTempSensorError	:= StatusTemperatureInput(X20AT4222_119.Status01, 3) OR NOT X20AT4222_119.ModuleOk;
	gInksInputs[4].iTemperatureRaw := X20AT4222_119.TempInput[4];
	gInksInputs[4].xTempSensorError	:= StatusTemperatureInput(X20AT4222_119.Status01, 4) OR NOT X20AT4222_119.ModuleOk;

	gBlockInputs[1].xModuleTemp02Ok	:= X20AT4222_120.ModuleOk;
	gInksInputs[5].iTemperatureRaw := X20AT4222_120.TempInput[1];
	gInksInputs[5].xTempSensorError	:= StatusTemperatureInput(X20AT4222_120.Status01, 1)  OR NOT X20AT4222_120.ModuleOk;

	// SI UNIT BK1
	gBlockInputs[1].xSiUnitModuleOk		:= SiUnitPwrLnkBK1.ModuleOk;
	gMachine.In.xAirSupply				:= SiUnitPwrLnkBK1.Input01_16.0;
	gBlockInputs[1].xAirVenturiOK		:= SiUnitPwrLnkBK1.Input01_16.1;
	gBlockInputs[1].xTrayOut			:= SiUnitPwrLnkBK1.Input01_16.2;
	gBlockInputs[1].xIclaSensor			:= SiUnitPwrLnkBK1.Input01_16.3;
	gTransVacuum[1].Inputs.xVaccAirFlow	:= SiUnitPwrLnkBK1.Input01_16.4;
	//SPARE 							:= SiUnitPwrLnkBK1.Input01_16.5;
	gBlockInputs[1].xBarsIn 			:= SiUnitPwrLnkBK1.Input01_16.6;

	gTransVacuum[1].Inputs.xSafetyEnable := gMachine.In.xSafetyEnabled; // NOTE: Check the order of assignation. This one after the machine one
	// := SiUnitPwrLnkBK1.Input01_16.7;

	//Signals Forced by Configuration
	gBlockInputs[1].Safety.xFrontEStopOK := TRUE;
	gBlockInputs[1].Safety.xRearEStopOK := TRUE;

	gBlockInputs[1].Safety.xFrontSafetyOK	:= TRUE;
	gBlockInputs[1].Safety.xRearSafetyOK	:= TRUE;
	gBlockInputs[1].Safety.xSafetyOK 		:= gMachine.In.xSafetyEnabled;

	//There are no light curtains so assigning the only safety outputs by safety controller
	gBlockInputs[1].Safety.xCurtainEnable01 := gBlockInputs[1].Safety.xCurtainEnable02 := TRUE;

	//Signals Forced by Configuration
	FOR iIndexVac := 1 TO MAX_LAST_TRANS_VACUUM DO gTransVacuum[iIndexVac].Inputs.xBlowersAnyCB := FALSE; END_FOR

	//Forcing some variable to TRUE so hardware required is not installed in this machine
	gBelt.parameters.xDriveProtectionOK := TRUE; //This machine has no feedback wired from electrical protection. An alternative is to check axis belt information about power supply
	gBlockInputs[1].xDriveProtectionOK := gBlockInputs[1].xDifferentialOK := TRUE;

	//Signals Forced by Configuration
	FOR iIndexBlock := 1 TO gMachine.Pt.CT.iNumBlocks DO
		gBlockInputs[iIndexBlock].xHeaterDcOkBusBar1 := TRUE;
		gBlockInputs[iIndexBlock].xHeaterDcOkBusBar2 := TRUE;

		gBlock[iIndexBlock].parameters.Hw.iNumPrintheadsPSU := 1;
		gBlock[iIndexBlock].parameters.Hw.iNumHeaterPSU := 1;
	END_FOR

END_ACTION
```
